// Mitsubishi GX Developer project: パレット移載装置   PLC: Q02

PROGRAM ALARM
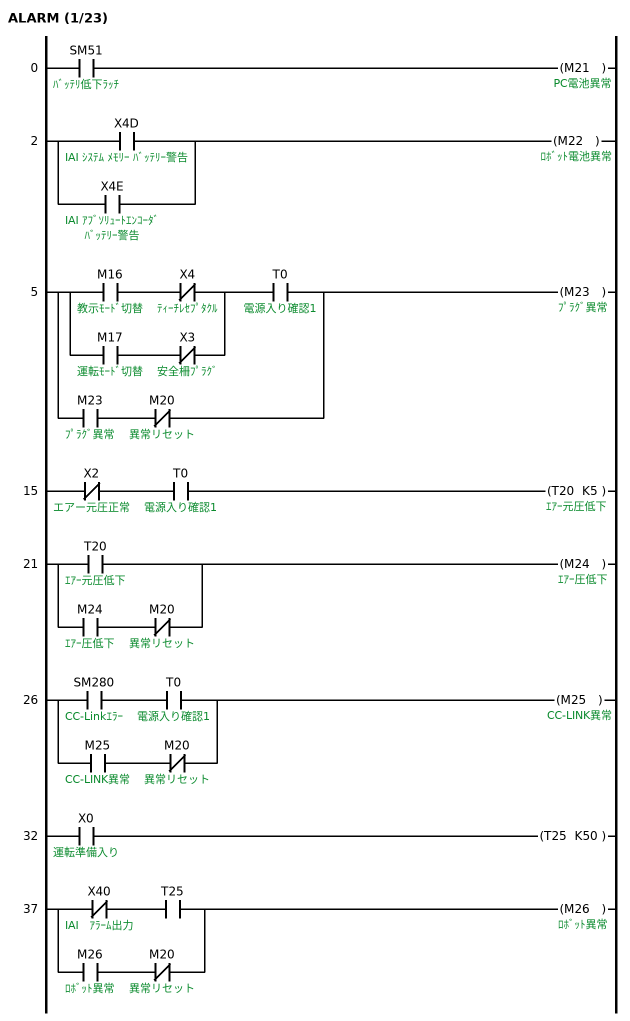
0     LD      SM51  ; ﾊﾞｯﾃﾘ低下ﾗｯﾁ
      OUT     M21  ; PC電池異常
2     LD      X4D  ; IAI ｼｽﾃﾑ ﾒﾓﾘｰ ﾊﾞｯﾃﾘｰ警告
      OR      X4E  ; IAI ｱﾌﾞｿﾘｭｰﾄｴﾝｺｰﾀﾞ ﾊﾞｯﾃﾘｰ警告
      OUT     M22  ; ﾛﾎﾞｯﾄ電池異常
5     LD      M16  ; 教示ﾓｰﾄﾞ切替
      ANI     X4  ; ﾃｨｰﾁﾚｾﾌﾟﾀｸﾙ
      LD      M17  ; 運転ﾓｰﾄﾞ切替
      ANI     X3  ; 安全柵ﾌﾟﾗｸﾞ
      ORB
      AND     T0  ; 電源入り確認1
      LD      M23  ; ﾌﾟﾗｸﾞ異常
      ANI     M20  ; 異常リセット
      ORB
      OUT     M23  ; ﾌﾟﾗｸﾞ異常
15    LDI     X2  ; エアー元圧正常
      AND     T0  ; 電源入り確認1
      OUT     T20 K5  ; ｴｱｰ元圧低下
21    LD      T20  ; ｴｱｰ元圧低下
      LD      M24  ; ｴｱｰ圧低下
      ANI     M20  ; 異常リセット
      ORB
      OUT     M24  ; ｴｱｰ圧低下
26    LD      SM280  ; CC-Linkｴﾗｰ
      AND     T0  ; 電源入り確認1
      LD      M25  ; CC-LINK異常
      ANI     M20  ; 異常リセット
      ORB
      OUT     M25  ; CC-LINK異常
32    LD      X0  ; 運転準備入り
      OUT     T25 K50
37    LDI     X40  ; IAI　ｱﾗｰﾑ出力
      AND     T25
      LD      M26  ; ﾛﾎﾞｯﾄ異常
      ANI     M20  ; 異常リセット
      ORB
      OUT     M26  ; ﾛﾎﾞｯﾄ異常
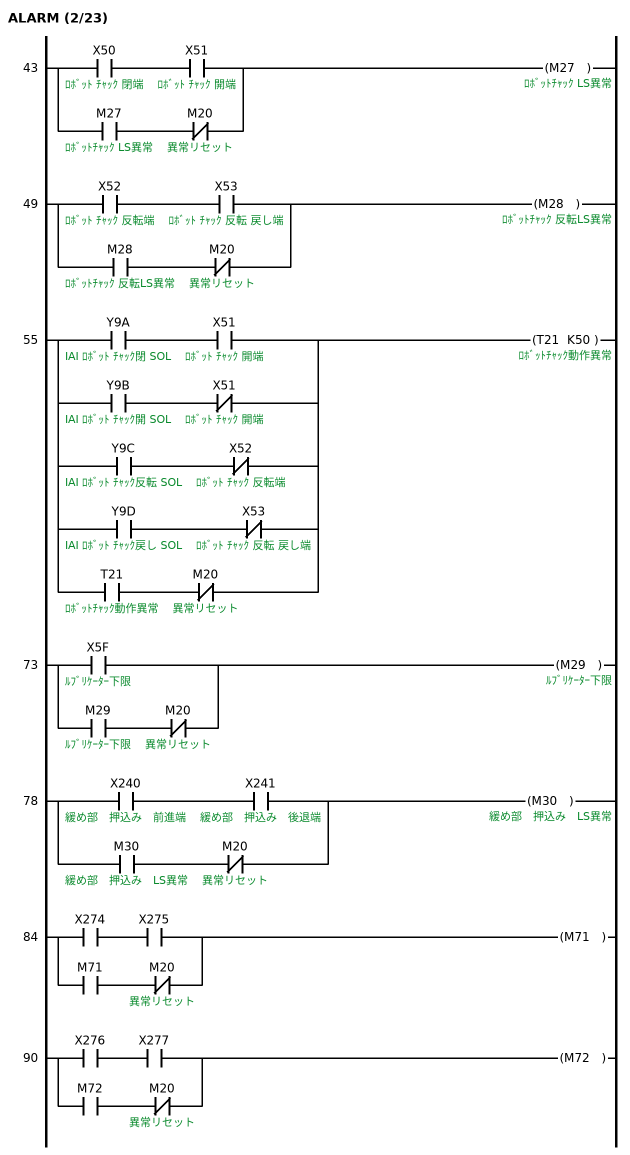
43    LD      X50  ; ﾛﾎﾞｯﾄ ﾁｬｯｸ 閉端
      AND     X51  ; ﾛﾎﾞｯﾄ ﾁｬｯｸ 開端
      LD      M27  ; ﾛﾎﾞｯﾄﾁｬｯｸ LS異常
      ANI     M20  ; 異常リセット
      ORB
      OUT     M27  ; ﾛﾎﾞｯﾄﾁｬｯｸ LS異常
49    LD      X52  ; ﾛﾎﾞｯﾄ ﾁｬｯｸ 反転端
      AND     X53  ; ﾛﾎﾞｯﾄ ﾁｬｯｸ 反転 戻し端
      LD      M28  ; ﾛﾎﾞｯﾄﾁｬｯｸ 反転LS異常
      ANI     M20  ; 異常リセット
      ORB
      OUT     M28  ; ﾛﾎﾞｯﾄﾁｬｯｸ 反転LS異常
55    LD      Y9A  ; IAI ﾛﾎﾞｯﾄ ﾁｬｯｸ閉 SOL
      AND     X51  ; ﾛﾎﾞｯﾄ ﾁｬｯｸ 開端
      LD      Y9B  ; IAI ﾛﾎﾞｯﾄ ﾁｬｯｸ開 SOL
      ANI     X51  ; ﾛﾎﾞｯﾄ ﾁｬｯｸ 開端
      ORB
      LD      Y9C  ; IAI ﾛﾎﾞｯﾄ ﾁｬｯｸ反転 SOL
      ANI     X52  ; ﾛﾎﾞｯﾄ ﾁｬｯｸ 反転端
      ORB
      LD      Y9D  ; IAI ﾛﾎﾞｯﾄ ﾁｬｯｸ戻し SOL
      ANI     X53  ; ﾛﾎﾞｯﾄ ﾁｬｯｸ 反転 戻し端
      ORB
      LD      T21  ; ﾛﾎﾞｯﾄﾁｬｯｸ動作異常
      ANI     M20  ; 異常リセット
      ORB
      OUT     T21 K50  ; ﾛﾎﾞｯﾄﾁｬｯｸ動作異常
73    LD      X5F  ; ﾙﾌﾞﾘｹｰﾀｰ下限
      LD      M29  ; ﾙﾌﾞﾘｹｰﾀｰ下限
      ANI     M20  ; 異常リセット
      ORB
      OUT     M29  ; ﾙﾌﾞﾘｹｰﾀｰ下限
78    LD      X240  ; 緩め部　押込み　前進端
      AND     X241  ; 緩め部　押込み　後退端
      LD      M30  ; 緩め部　押込み　LS異常
      ANI     M20  ; 異常リセット
      ORB
      OUT     M30  ; 緩め部　押込み　LS異常
84    LD      X274
      AND     X275
      LD      M71
      ANI     M20  ; 異常リセット
      ORB
      OUT     M71
90    LD      X276
      AND     X277
      LD      M72
      ANI     M20  ; 異常リセット
      ORB
      OUT     M72
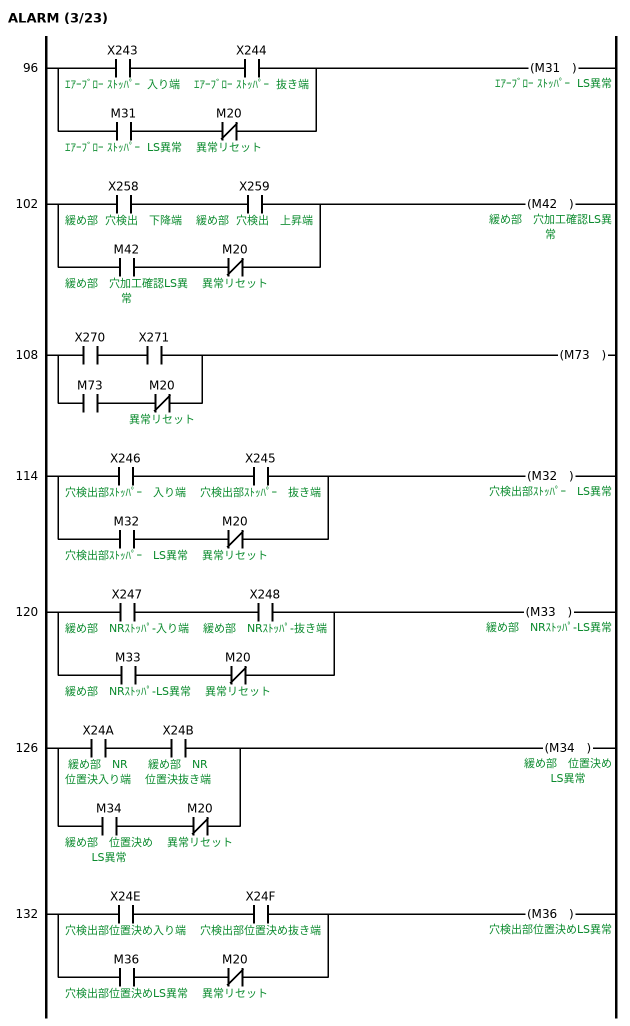
96    LD      X243  ; ｴｱｰﾌﾞﾛｰ ｽﾄｯﾊﾟｰ  入り端
      AND     X244  ; ｴｱｰﾌﾞﾛｰ ｽﾄｯﾊﾟｰ  抜き端
      LD      M31  ; ｴｱｰﾌﾞﾛｰ ｽﾄｯﾊﾟｰ  LS異常
      ANI     M20  ; 異常リセット
      ORB
      OUT     M31  ; ｴｱｰﾌﾞﾛｰ ｽﾄｯﾊﾟｰ  LS異常
102   LD      X258  ; 緩め部  穴検出　下降端
      AND     X259  ; 緩め部  穴検出　上昇端
      LD      M42  ; 緩め部　穴加工確認LS異常
      ANI     M20  ; 異常リセット
      ORB
      OUT     M42  ; 緩め部　穴加工確認LS異常
108   LD      X270
      AND     X271
      LD      M73
      ANI     M20  ; 異常リセット
      ORB
      OUT     M73
114   LD      X246  ; 穴検出部ｽﾄｯﾊﾟｰ　入り端
      AND     X245  ; 穴検出部ｽﾄｯﾊﾟｰ　抜き端
      LD      M32  ; 穴検出部ｽﾄｯﾊﾟｰ　LS異常
      ANI     M20  ; 異常リセット
      ORB
      OUT     M32  ; 穴検出部ｽﾄｯﾊﾟｰ　LS異常
120   LD      X247  ; 緩め部　NRｽﾄｯﾊﾟ-入り端
      AND     X248  ; 緩め部　NRｽﾄｯﾊﾟ-抜き端
      LD      M33  ; 緩め部　NRｽﾄｯﾊﾟ-LS異常
      ANI     M20  ; 異常リセット
      ORB
      OUT     M33  ; 緩め部　NRｽﾄｯﾊﾟ-LS異常
126   LD      X24A  ; 緩め部　NR 位置決入り端
      AND     X24B  ; 緩め部　NR 位置決抜き端
      LD      M34  ; 緩め部　位置決め LS異常
      ANI     M20  ; 異常リセット
      ORB
      OUT     M34  ; 緩め部　位置決め LS異常
132   LD      X24E  ; 穴検出部位置決め入り端
      AND     X24F  ; 穴検出部位置決め抜き端
      LD      M36  ; 穴検出部位置決めLS異常
      ANI     M20  ; 異常リセット
      ORB
      OUT     M36  ; 穴検出部位置決めLS異常
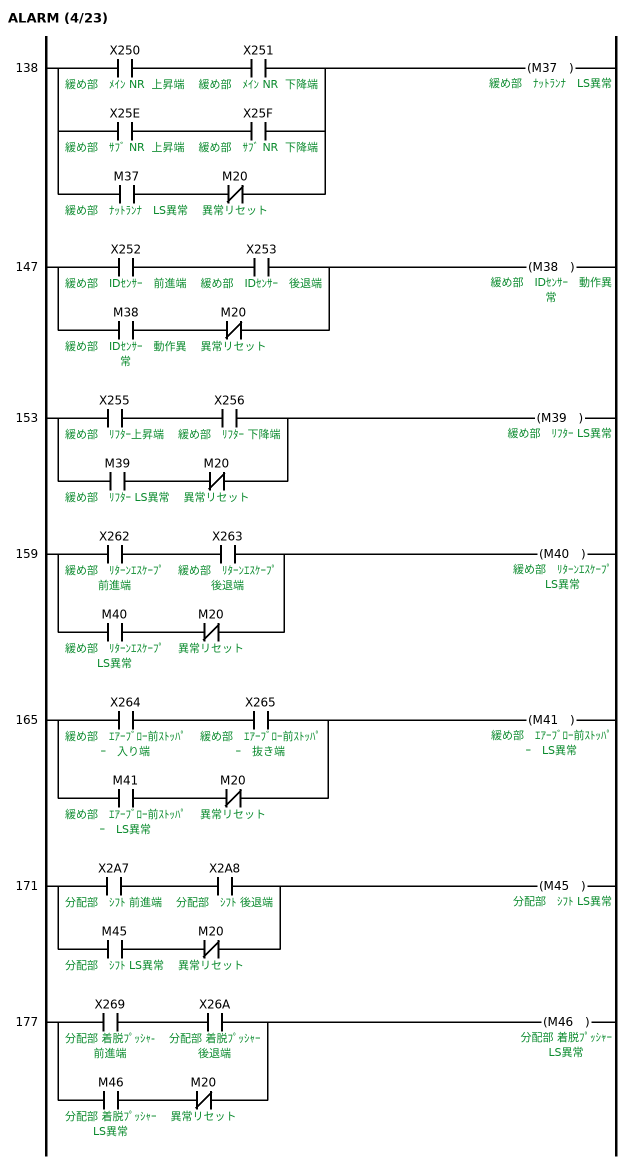
138   LD      X250  ; 緩め部　ﾒｲﾝ NR  上昇端
      AND     X251  ; 緩め部　ﾒｲﾝ NR  下降端
      LD      X25E  ; 緩め部　ｻﾌﾞ NR  上昇端
      AND     X25F  ; 緩め部　ｻﾌﾞ NR  下降端
      ORB
      LD      M37  ; 緩め部　ﾅｯﾄﾗﾝﾅ　LS異常
      ANI     M20  ; 異常リセット
      ORB
      OUT     M37  ; 緩め部　ﾅｯﾄﾗﾝﾅ　LS異常
147   LD      X252  ; 緩め部　IDｾﾝｻｰ　前進端
      AND     X253  ; 緩め部　IDｾﾝｻｰ　後退端
      LD      M38  ; 緩め部　IDｾﾝｻｰ　動作異常
      ANI     M20  ; 異常リセット
      ORB
      OUT     M38  ; 緩め部　IDｾﾝｻｰ　動作異常
153   LD      X255  ; 緩め部　ﾘﾌﾀｰ上昇端
      AND     X256  ; 緩め部　ﾘﾌﾀｰ 下降端
      LD      M39  ; 緩め部　ﾘﾌﾀｰ LS異常
      ANI     M20  ; 異常リセット
      ORB
      OUT     M39  ; 緩め部　ﾘﾌﾀｰ LS異常
159   LD      X262  ; 緩め部　ﾘﾀｰﾝｴｽｹｰﾌﾟ 前進端
      AND     X263  ; 緩め部　ﾘﾀｰﾝｴｽｹｰﾌﾟ 後退端
      LD      M40  ; 緩め部　ﾘﾀｰﾝｴｽｹｰﾌﾟ LS異常
      ANI     M20  ; 異常リセット
      ORB
      OUT     M40  ; 緩め部　ﾘﾀｰﾝｴｽｹｰﾌﾟ LS異常
165   LD      X264  ; 緩め部　ｴｱｰﾌﾞﾛｰ前ｽﾄｯﾊﾟｰ　入り端
      AND     X265  ; 緩め部　ｴｱｰﾌﾞﾛｰ前ｽﾄｯﾊﾟｰ　抜き端
      LD      M41  ; 緩め部　ｴｱｰﾌﾞﾛｰ前ｽﾄｯﾊﾟｰ　LS異常
      ANI     M20  ; 異常リセット
      ORB
      OUT     M41  ; 緩め部　ｴｱｰﾌﾞﾛｰ前ｽﾄｯﾊﾟｰ　LS異常
171   LD      X2A7  ; 分配部　ｼﾌﾄ 前進端
      AND     X2A8  ; 分配部　ｼﾌﾄ 後退端
      LD      M45  ; 分配部　ｼﾌﾄ LS異常
      ANI     M20  ; 異常リセット
      ORB
      OUT     M45  ; 分配部　ｼﾌﾄ LS異常
177   LD      X269  ; 分配部 着脱ﾌﾟｯｼｬ- 前進端
      AND     X26A  ; 分配部 着脱ﾌﾟｯｼｬｰ 後退端
      LD      M46  ; 分配部 着脱ﾌﾟｯｼｬｰ LS異常
      ANI     M20  ; 異常リセット
      ORB
      OUT     M46  ; 分配部 着脱ﾌﾟｯｼｬｰ LS異常
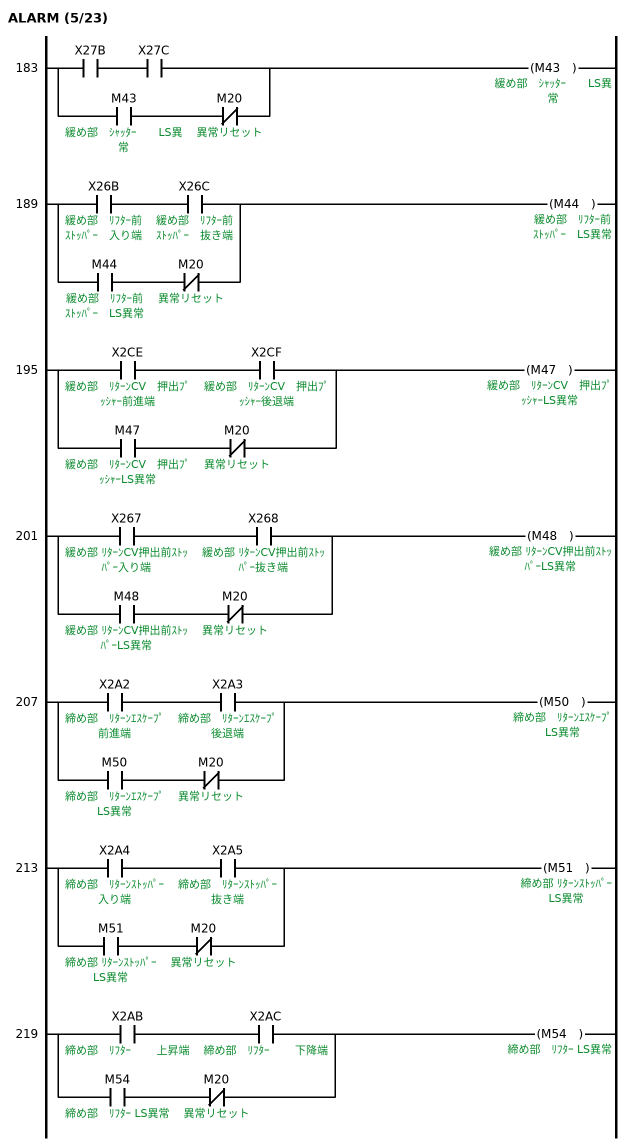
183   LD      X27B
      AND     X27C
      LD      M43  ; 緩め部　ｼｬｯﾀｰ　　LS異常
      ANI     M20  ; 異常リセット
      ORB
      OUT     M43  ; 緩め部　ｼｬｯﾀｰ　　LS異常
189   LD      X26B  ; 緩め部　ﾘﾌﾀｰ前  ｽﾄｯﾊﾟｰ　入り端
      AND     X26C  ; 緩め部　ﾘﾌﾀｰ前  ｽﾄｯﾊﾟｰ　抜き端
      LD      M44  ; 緩め部　ﾘﾌﾀｰ前  ｽﾄｯﾊﾟｰ　LS異常
      ANI     M20  ; 異常リセット
      ORB
      OUT     M44  ; 緩め部　ﾘﾌﾀｰ前  ｽﾄｯﾊﾟｰ　LS異常
195   LD      X2CE  ; 緩め部　ﾘﾀｰﾝCV　押出ﾌﾟｯｼｬｰ前進端
      AND     X2CF  ; 緩め部　ﾘﾀｰﾝCV　押出ﾌﾟｯｼｬｰ後退端
      LD      M47  ; 緩め部　ﾘﾀｰﾝCV　押出ﾌﾟｯｼｬｰLS異常
      ANI     M20  ; 異常リセット
      ORB
      OUT     M47  ; 緩め部　ﾘﾀｰﾝCV　押出ﾌﾟｯｼｬｰLS異常
201   LD      X267  ; 緩め部 ﾘﾀｰﾝCV押出前ｽﾄｯﾊﾟｰ入り端
      AND     X268  ; 緩め部 ﾘﾀｰﾝCV押出前ｽﾄｯﾊﾟｰ抜き端
      LD      M48  ; 緩め部 ﾘﾀｰﾝCV押出前ｽﾄｯﾊﾟｰLS異常
      ANI     M20  ; 異常リセット
      ORB
      OUT     M48  ; 緩め部 ﾘﾀｰﾝCV押出前ｽﾄｯﾊﾟｰLS異常
207   LD      X2A2  ; 締め部　ﾘﾀｰﾝｴｽｹｰﾌﾟ 前進端
      AND     X2A3  ; 締め部　ﾘﾀｰﾝｴｽｹｰﾌﾟ 後退端
      LD      M50  ; 締め部　ﾘﾀｰﾝｴｽｹｰﾌﾟ LS異常
      ANI     M20  ; 異常リセット
      ORB
      OUT     M50  ; 締め部　ﾘﾀｰﾝｴｽｹｰﾌﾟ LS異常
213   LD      X2A4  ; 締め部　ﾘﾀｰﾝｽﾄｯﾊﾟｰ 入り端
      AND     X2A5  ; 締め部　ﾘﾀｰﾝｽﾄｯﾊﾟｰ 抜き端
      LD      M51  ; 締め部 ﾘﾀｰﾝｽﾄｯﾊﾟｰ LS異常
      ANI     M20  ; 異常リセット
      ORB
      OUT     M51  ; 締め部 ﾘﾀｰﾝｽﾄｯﾊﾟｰ LS異常
219   LD      X2AB  ; 締め部　ﾘﾌﾀｰ 　　上昇端
      AND     X2AC  ; 締め部　ﾘﾌﾀｰ 　　下降端
      LD      M54  ; 締め部　ﾘﾌﾀｰ LS異常
      ANI     M20  ; 異常リセット
      ORB
      OUT     M54  ; 締め部　ﾘﾌﾀｰ LS異常
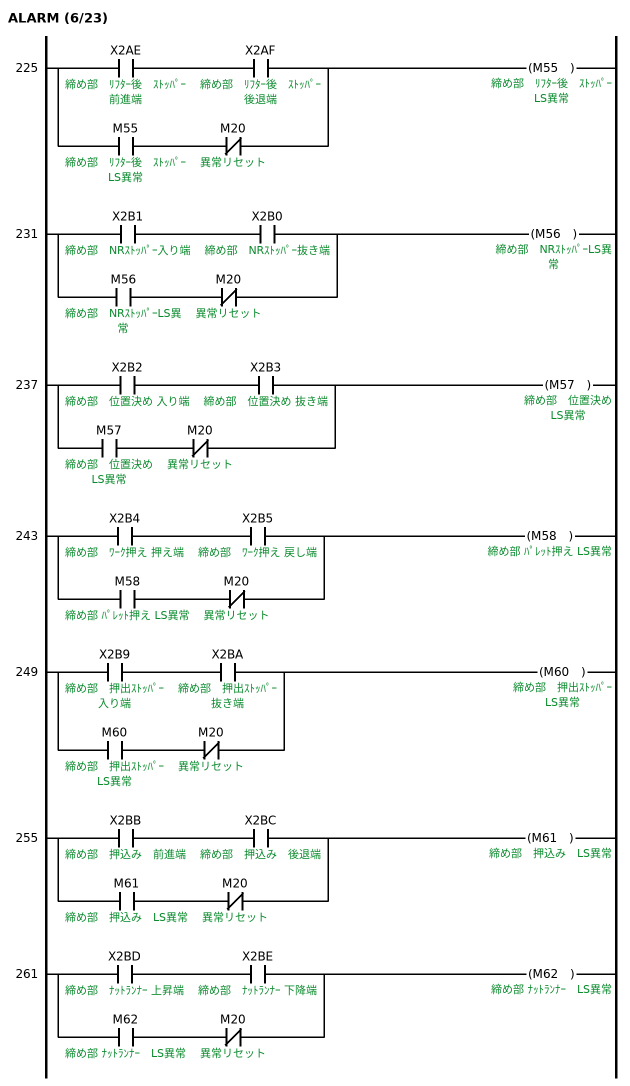
225   LD      X2AE  ; 締め部　ﾘﾌﾀｰ後　ｽﾄｯﾊﾟｰ　前進端
      AND     X2AF  ; 締め部　ﾘﾌﾀｰ後　ｽﾄｯﾊﾟｰ　後退端
      LD      M55  ; 締め部　ﾘﾌﾀｰ後　ｽﾄｯﾊﾟｰ　LS異常
      ANI     M20  ; 異常リセット
      ORB
      OUT     M55  ; 締め部　ﾘﾌﾀｰ後　ｽﾄｯﾊﾟｰ　LS異常
231   LD      X2B1  ; 締め部　NRｽﾄｯﾊﾟｰ入り端
      AND     X2B0  ; 締め部　NRｽﾄｯﾊﾟｰ抜き端
      LD      M56  ; 締め部　NRｽﾄｯﾊﾟｰLS異常
      ANI     M20  ; 異常リセット
      ORB
      OUT     M56  ; 締め部　NRｽﾄｯﾊﾟｰLS異常
237   LD      X2B2  ; 締め部　位置決め 入り端
      AND     X2B3  ; 締め部　位置決め 抜き端
      LD      M57  ; 締め部　位置決め LS異常
      ANI     M20  ; 異常リセット
      ORB
      OUT     M57  ; 締め部　位置決め LS異常
243   LD      X2B4  ; 締め部　ﾜｰｸ押え 押え端
      AND     X2B5  ; 締め部　ﾜｰｸ押え 戻し端
      LD      M58  ; 締め部 ﾊﾟﾚｯﾄ押え LS異常
      ANI     M20  ; 異常リセット
      ORB
      OUT     M58  ; 締め部 ﾊﾟﾚｯﾄ押え LS異常
249   LD      X2B9  ; 締め部　押出ｽﾄｯﾊﾟｰ 入り端
      AND     X2BA  ; 締め部　押出ｽﾄｯﾊﾟｰ 抜き端
      LD      M60  ; 締め部　押出ｽﾄｯﾊﾟｰ LS異常
      ANI     M20  ; 異常リセット
      ORB
      OUT     M60  ; 締め部　押出ｽﾄｯﾊﾟｰ LS異常
255   LD      X2BB  ; 締め部　押込み　前進端
      AND     X2BC  ; 締め部　押込み　後退端
      LD      M61  ; 締め部　押込み　LS異常
      ANI     M20  ; 異常リセット
      ORB
      OUT     M61  ; 締め部　押込み　LS異常
261   LD      X2BD  ; 締め部　ﾅｯﾄﾗﾝﾅｰ 上昇端
      AND     X2BE  ; 締め部　ﾅｯﾄﾗﾝﾅｰ 下降端
      LD      M62  ; 締め部 ﾅｯﾄﾗﾝﾅｰ　LS異常
      ANI     M20  ; 異常リセット
      ORB
      OUT     M62  ; 締め部 ﾅｯﾄﾗﾝﾅｰ　LS異常
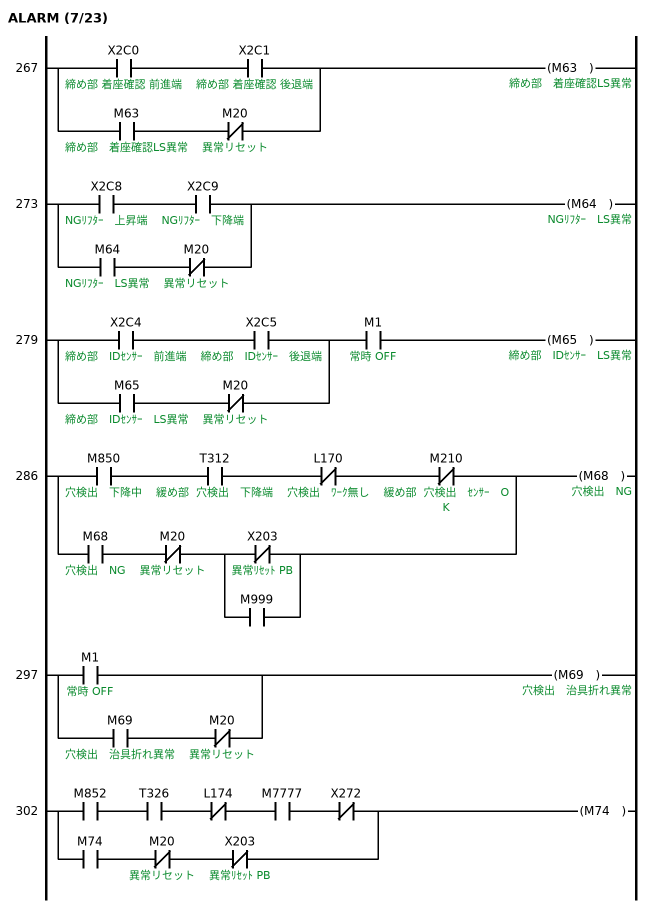
267   LD      X2C0  ; 締め部 着座確認 前進端
      AND     X2C1  ; 締め部 着座確認 後退端
      LD      M63  ; 締め部　着座確認LS異常
      ANI     M20  ; 異常リセット
      ORB
      OUT     M63  ; 締め部　着座確認LS異常
273   LD      X2C8  ; NGﾘﾌﾀｰ　上昇端
      AND     X2C9  ; NGﾘﾌﾀｰ　下降端
      LD      M64  ; NGﾘﾌﾀｰ　LS異常
      ANI     M20  ; 異常リセット
      ORB
      OUT     M64  ; NGﾘﾌﾀｰ　LS異常
279   LD      X2C4  ; 締め部　IDｾﾝｻｰ　前進端
      AND     X2C5  ; 締め部　IDｾﾝｻｰ　後退端
      LD      M65  ; 締め部　IDｾﾝｻｰ　LS異常
      ANI     M20  ; 異常リセット
      ORB
      AND     M1  ; 常時 OFF
      OUT     M65  ; 締め部　IDｾﾝｻｰ　LS異常
286   LD      M850  ; 穴検出　下降中
      AND     T312  ; 緩め部  穴検出　下降端
      ANI     L170  ; 穴検出　ﾜｰｸ無し
      ANI     M210  ; 緩め部  穴検出　ｾﾝｻｰ　OK
      LD      M68  ; 穴検出　NG
      ANI     M20  ; 異常リセット
      LDI     X203  ; 異常ﾘｾｯﾄ PB
      OR      M999
      ANB
      ORB
      OUT     M68  ; 穴検出　NG
297   LD      M1  ; 常時 OFF
      LD      M69  ; 穴検出　治具折れ異常
      ANI     M20  ; 異常リセット
      ORB
      OUT     M69  ; 穴検出　治具折れ異常
302   LD      M852
      AND     T326
      ANI     L174
      AND     M7777
      ANI     X272
      LD      M74
      ANI     M20  ; 異常リセット
      ANI     X203  ; 異常ﾘｾｯﾄ PB
      ORB
      OUT     M74
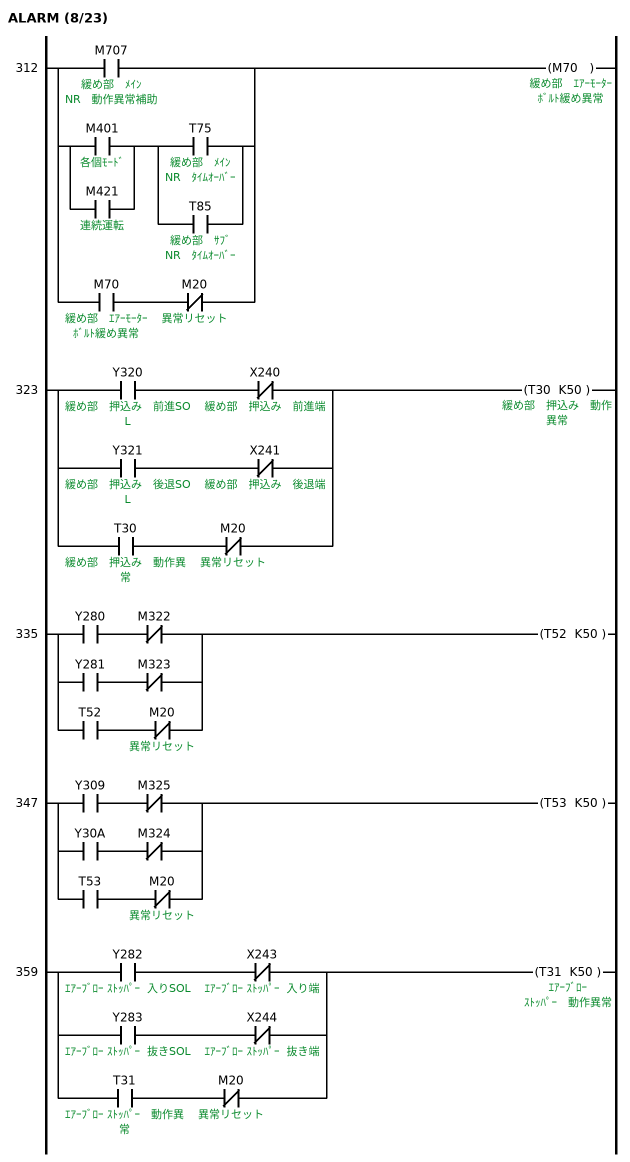
312   LD      M707  ; 緩め部　ﾒｲﾝ NR　動作異常補助
      LD      M401  ; 各個ﾓｰﾄﾞ
      OR      M421  ; 連続運転
      LD      T75  ; 緩め部　ﾒｲﾝ NR　ﾀｲﾑｵｰﾊﾞｰ
      OR      T85  ; 緩め部　ｻﾌﾞ NR　ﾀｲﾑｵｰﾊﾞｰ
      ANB
      ORB
      LD      M70  ; 緩め部　ｴｱｰﾓｰﾀｰ ﾎﾞﾙﾄ緩め異常
      ANI     M20  ; 異常リセット
      ORB
      OUT     M70  ; 緩め部　ｴｱｰﾓｰﾀｰ ﾎﾞﾙﾄ緩め異常
323   LD      Y320  ; 緩め部　押込み　前進SOL
      ANI     X240  ; 緩め部　押込み　前進端
      LD      Y321  ; 緩め部　押込み　後退SOL
      ANI     X241  ; 緩め部　押込み　後退端
      ORB
      LD      T30  ; 緩め部　押込み　動作異常
      ANI     M20  ; 異常リセット
      ORB
      OUT     T30 K50  ; 緩め部　押込み　動作異常
335   LD      Y280
      ANI     M322
      LD      Y281
      ANI     M323
      ORB
      LD      T52
      ANI     M20  ; 異常リセット
      ORB
      OUT     T52 K50
347   LD      Y309
      ANI     M325
      LD      Y30A
      ANI     M324
      ORB
      LD      T53
      ANI     M20  ; 異常リセット
      ORB
      OUT     T53 K50
359   LD      Y282  ; ｴｱｰﾌﾞﾛｰ ｽﾄｯﾊﾟｰ  入りSOL
      ANI     X243  ; ｴｱｰﾌﾞﾛｰ ｽﾄｯﾊﾟｰ  入り端
      LD      Y283  ; ｴｱｰﾌﾞﾛｰ ｽﾄｯﾊﾟｰ  抜きSOL
      ANI     X244  ; ｴｱｰﾌﾞﾛｰ ｽﾄｯﾊﾟｰ  抜き端
      ORB
      LD      T31  ; ｴｱｰﾌﾞﾛｰ ｽﾄｯﾊﾟｰ　動作異常
      ANI     M20  ; 異常リセット
      ORB
      OUT     T31 K50  ; ｴｱｰﾌﾞﾛｰ ｽﾄｯﾊﾟｰ　動作異常
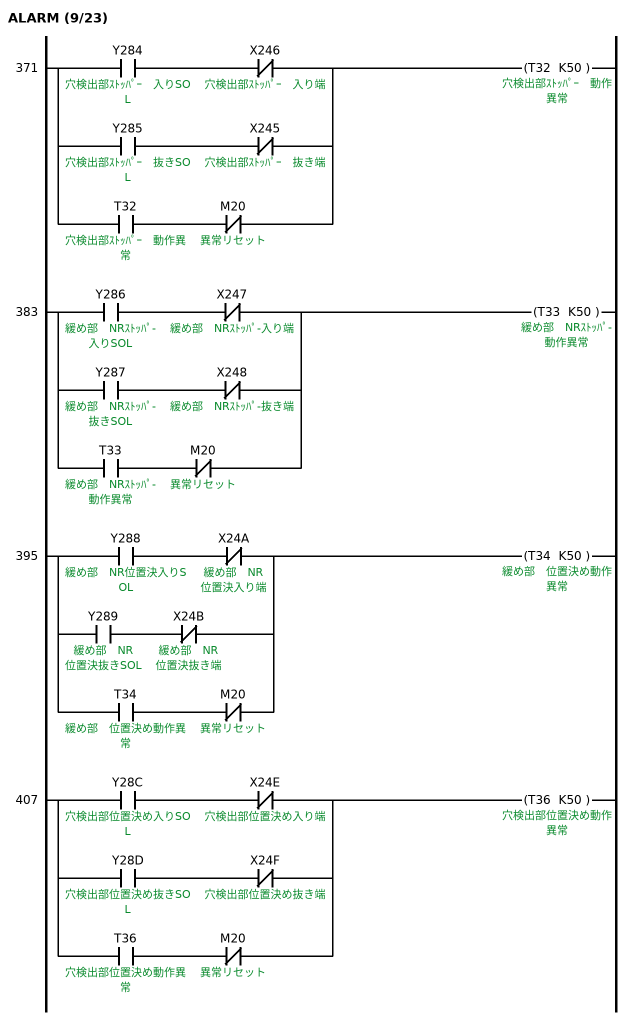
371   LD      Y284  ; 穴検出部ｽﾄｯﾊﾟｰ　入りSOL
      ANI     X246  ; 穴検出部ｽﾄｯﾊﾟｰ　入り端
      LD      Y285  ; 穴検出部ｽﾄｯﾊﾟｰ　抜きSOL
      ANI     X245  ; 穴検出部ｽﾄｯﾊﾟｰ　抜き端
      ORB
      LD      T32  ; 穴検出部ｽﾄｯﾊﾟｰ　動作異常
      ANI     M20  ; 異常リセット
      ORB
      OUT     T32 K50  ; 穴検出部ｽﾄｯﾊﾟｰ　動作異常
383   LD      Y286  ; 緩め部　NRｽﾄｯﾊﾟ-入りSOL
      ANI     X247  ; 緩め部　NRｽﾄｯﾊﾟ-入り端
      LD      Y287  ; 緩め部　NRｽﾄｯﾊﾟ-抜きSOL
      ANI     X248  ; 緩め部　NRｽﾄｯﾊﾟ-抜き端
      ORB
      LD      T33  ; 緩め部　NRｽﾄｯﾊﾟ-動作異常
      ANI     M20  ; 異常リセット
      ORB
      OUT     T33 K50  ; 緩め部　NRｽﾄｯﾊﾟ-動作異常
395   LD      Y288  ; 緩め部　NR位置決入りSOL
      ANI     X24A  ; 緩め部　NR 位置決入り端
      LD      Y289  ; 緩め部　NR 位置決抜きSOL
      ANI     X24B  ; 緩め部　NR 位置決抜き端
      ORB
      LD      T34  ; 緩め部　位置決め動作異常
      ANI     M20  ; 異常リセット
      ORB
      OUT     T34 K50  ; 緩め部　位置決め動作異常
407   LD      Y28C  ; 穴検出部位置決め入りSOL
      ANI     X24E  ; 穴検出部位置決め入り端
      LD      Y28D  ; 穴検出部位置決め抜きSOL
      ANI     X24F  ; 穴検出部位置決め抜き端
      ORB
      LD      T36  ; 穴検出部位置決め動作異常
      ANI     M20  ; 異常リセット
      ORB
      OUT     T36 K50  ; 穴検出部位置決め動作異常
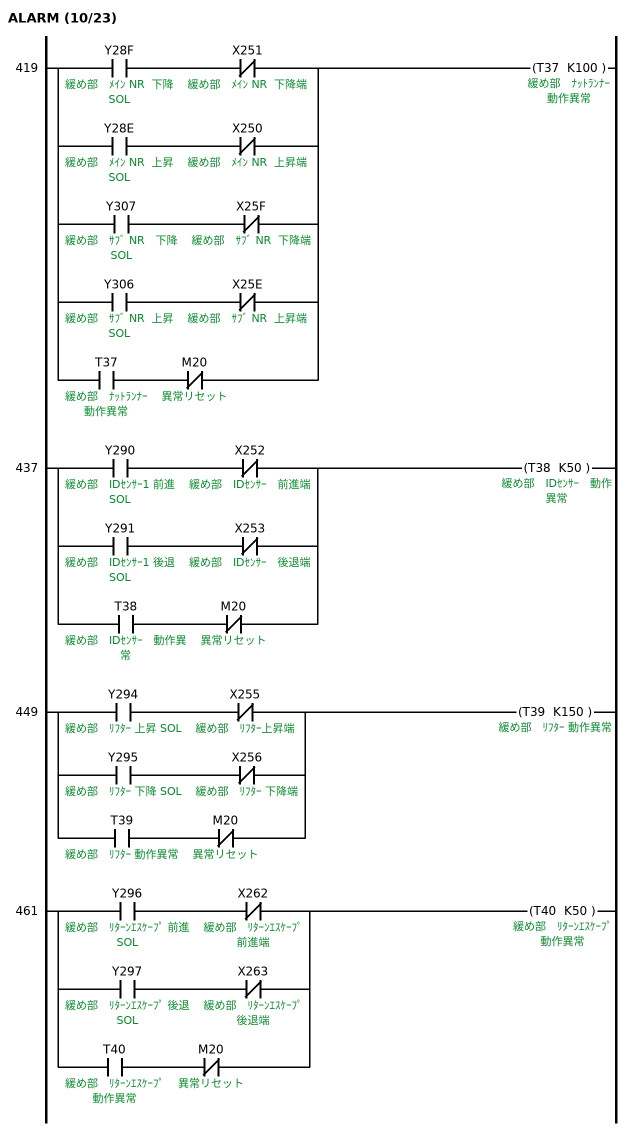
419   LD      Y28F  ; 緩め部　ﾒｲﾝ NR  下降 SOL
      ANI     X251  ; 緩め部　ﾒｲﾝ NR  下降端
      LD      Y28E  ; 緩め部　ﾒｲﾝ NR  上昇 SOL
      ANI     X250  ; 緩め部　ﾒｲﾝ NR  上昇端
      ORB
      LD      Y307  ; 緩め部　ｻﾌﾞ NR　下降 SOL
      ANI     X25F  ; 緩め部　ｻﾌﾞ NR  下降端
      ORB
      LD      Y306  ; 緩め部　ｻﾌﾞ NR  上昇 SOL
      ANI     X25E  ; 緩め部　ｻﾌﾞ NR  上昇端
      ORB
      LD      T37  ; 緩め部　ﾅｯﾄﾗﾝﾅｰ 動作異常
      ANI     M20  ; 異常リセット
      ORB
      OUT     T37 K100  ; 緩め部　ﾅｯﾄﾗﾝﾅｰ 動作異常
437   LD      Y290  ; 緩め部　IDｾﾝｻｰ1 前進 SOL
      ANI     X252  ; 緩め部　IDｾﾝｻｰ　前進端
      LD      Y291  ; 緩め部　IDｾﾝｻｰ1 後退 SOL
      ANI     X253  ; 緩め部　IDｾﾝｻｰ　後退端
      ORB
      LD      T38  ; 緩め部　IDｾﾝｻｰ　動作異常
      ANI     M20  ; 異常リセット
      ORB
      OUT     T38 K50  ; 緩め部　IDｾﾝｻｰ　動作異常
449   LD      Y294  ; 緩め部　ﾘﾌﾀｰ 上昇 SOL
      ANI     X255  ; 緩め部　ﾘﾌﾀｰ上昇端
      LD      Y295  ; 緩め部　ﾘﾌﾀｰ 下降 SOL
      ANI     X256  ; 緩め部　ﾘﾌﾀｰ 下降端
      ORB
      LD      T39  ; 緩め部　ﾘﾌﾀｰ 動作異常
      ANI     M20  ; 異常リセット
      ORB
      OUT     T39 K150  ; 緩め部　ﾘﾌﾀｰ 動作異常
461   LD      Y296  ; 緩め部　ﾘﾀｰﾝｴｽｹｰﾌﾟ 前進 SOL
      ANI     X262  ; 緩め部　ﾘﾀｰﾝｴｽｹｰﾌﾟ 前進端
      LD      Y297  ; 緩め部　ﾘﾀｰﾝｴｽｹｰﾌﾟ 後退 SOL
      ANI     X263  ; 緩め部　ﾘﾀｰﾝｴｽｹｰﾌﾟ 後退端
      ORB
      LD      T40  ; 緩め部　ﾘﾀｰﾝｴｽｹｰﾌﾟ 動作異常
      ANI     M20  ; 異常リセット
      ORB
      OUT     T40 K50  ; 緩め部　ﾘﾀｰﾝｴｽｹｰﾌﾟ 動作異常
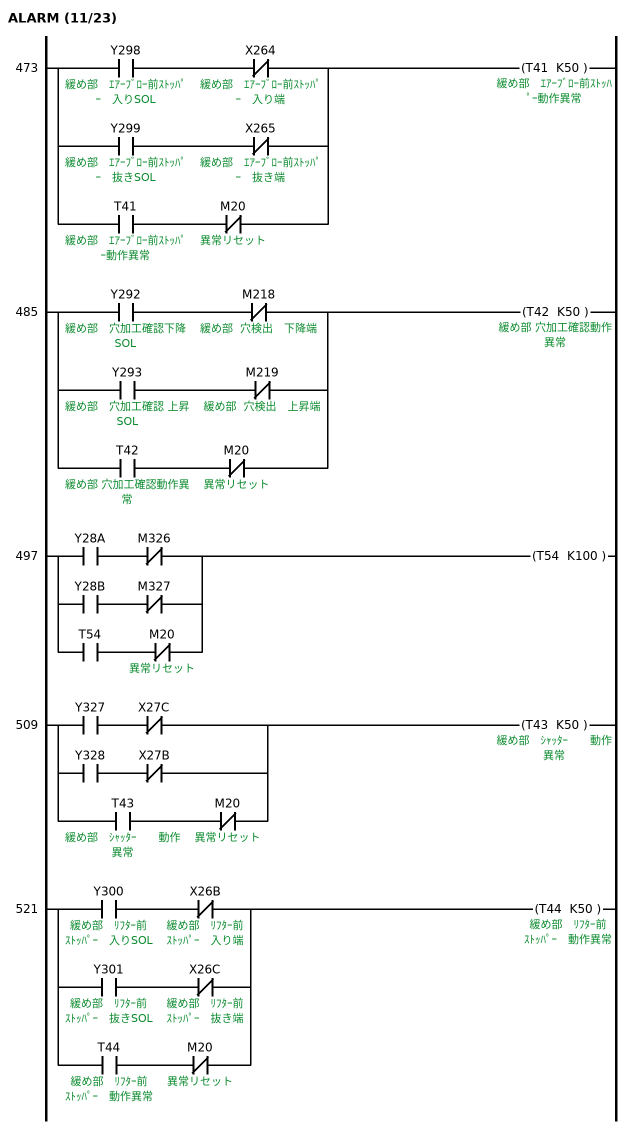
473   LD      Y298  ; 緩め部　ｴｱｰﾌﾞﾛｰ前ｽﾄｯﾊﾟｰ　入りSOL
      ANI     X264  ; 緩め部　ｴｱｰﾌﾞﾛｰ前ｽﾄｯﾊﾟｰ　入り端
      LD      Y299  ; 緩め部　ｴｱｰﾌﾞﾛｰ前ｽﾄｯﾊﾟｰ　抜きSOL
      ANI     X265  ; 緩め部　ｴｱｰﾌﾞﾛｰ前ｽﾄｯﾊﾟｰ　抜き端
      ORB
      LD      T41  ; 緩め部　ｴｱｰﾌﾞﾛｰ前ｽﾄｯﾊﾟｰ動作異常
      ANI     M20  ; 異常リセット
      ORB
      OUT     T41 K50  ; 緩め部　ｴｱｰﾌﾞﾛｰ前ｽﾄｯﾊﾟｰ動作異常
485   LD      Y292  ; 緩め部　穴加工確認下降 SOL
      ANI     M218  ; 緩め部  穴検出　下降端
      LD      Y293  ; 緩め部　穴加工確認 上昇 SOL
      ANI     M219  ; 緩め部  穴検出　上昇端
      ORB
      LD      T42  ; 緩め部 穴加工確認動作異常
      ANI     M20  ; 異常リセット
      ORB
      OUT     T42 K50  ; 緩め部 穴加工確認動作異常
497   LD      Y28A
      ANI     M326
      LD      Y28B
      ANI     M327
      ORB
      LD      T54
      ANI     M20  ; 異常リセット
      ORB
      OUT     T54 K100
509   LD      Y327
      ANI     X27C
      LD      Y328
      ANI     X27B
      ORB
      LD      T43  ; 緩め部　ｼｬｯﾀｰ　　動作異常
      ANI     M20  ; 異常リセット
      ORB
      OUT     T43 K50  ; 緩め部　ｼｬｯﾀｰ　　動作異常
521   LD      Y300  ; 緩め部　ﾘﾌﾀｰ前  ｽﾄｯﾊﾟｰ　入りSOL
      ANI     X26B  ; 緩め部　ﾘﾌﾀｰ前  ｽﾄｯﾊﾟｰ　入り端
      LD      Y301  ; 緩め部　ﾘﾌﾀｰ前  ｽﾄｯﾊﾟｰ　抜きSOL
      ANI     X26C  ; 緩め部　ﾘﾌﾀｰ前  ｽﾄｯﾊﾟｰ　抜き端
      ORB
      LD      T44  ; 緩め部　ﾘﾌﾀｰ前  ｽﾄｯﾊﾟｰ　動作異常
      ANI     M20  ; 異常リセット
      ORB
      OUT     T44 K50  ; 緩め部　ﾘﾌﾀｰ前  ｽﾄｯﾊﾟｰ　動作異常
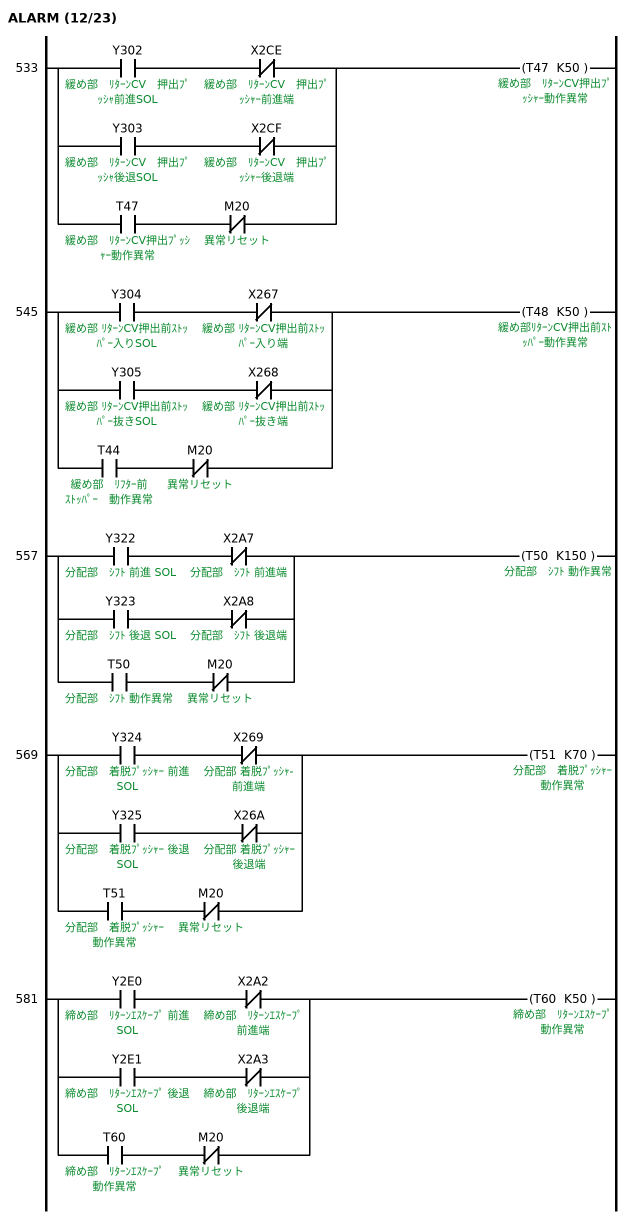
533   LD      Y302  ; 緩め部　ﾘﾀｰﾝCV　押出ﾌﾟｯｼｬ前進SOL
      ANI     X2CE  ; 緩め部　ﾘﾀｰﾝCV　押出ﾌﾟｯｼｬｰ前進端
      LD      Y303  ; 緩め部　ﾘﾀｰﾝCV　押出ﾌﾟｯｼｬ後退SOL
      ANI     X2CF  ; 緩め部　ﾘﾀｰﾝCV　押出ﾌﾟｯｼｬｰ後退端
      ORB
      LD      T47  ; 緩め部　ﾘﾀｰﾝCV押出ﾌﾟｯｼｬｰ動作異常
      ANI     M20  ; 異常リセット
      ORB
      OUT     T47 K50  ; 緩め部　ﾘﾀｰﾝCV押出ﾌﾟｯｼｬｰ動作異常
545   LD      Y304  ; 緩め部 ﾘﾀｰﾝCV押出前ｽﾄｯﾊﾟｰ入りSOL
      ANI     X267  ; 緩め部 ﾘﾀｰﾝCV押出前ｽﾄｯﾊﾟｰ入り端
      LD      Y305  ; 緩め部 ﾘﾀｰﾝCV押出前ｽﾄｯﾊﾟｰ抜きSOL
      ANI     X268  ; 緩め部 ﾘﾀｰﾝCV押出前ｽﾄｯﾊﾟｰ抜き端
      ORB
      LD      T44  ; 緩め部　ﾘﾌﾀｰ前  ｽﾄｯﾊﾟｰ　動作異常
      ANI     M20  ; 異常リセット
      ORB
      OUT     T48 K50  ; 緩め部ﾘﾀｰﾝCV押出前ｽﾄｯﾊﾟｰ動作異常
557   LD      Y322  ; 分配部　ｼﾌﾄ 前進 SOL
      ANI     X2A7  ; 分配部　ｼﾌﾄ 前進端
      LD      Y323  ; 分配部　ｼﾌﾄ 後退 SOL
      ANI     X2A8  ; 分配部　ｼﾌﾄ 後退端
      ORB
      LD      T50  ; 分配部　ｼﾌﾄ 動作異常
      ANI     M20  ; 異常リセット
      ORB
      OUT     T50 K150  ; 分配部　ｼﾌﾄ 動作異常
569   LD      Y324  ; 分配部　着脱ﾌﾟｯｼｬｰ 前進 SOL
      ANI     X269  ; 分配部 着脱ﾌﾟｯｼｬ- 前進端
      LD      Y325  ; 分配部　着脱ﾌﾟｯｼｬｰ 後退 SOL
      ANI     X26A  ; 分配部 着脱ﾌﾟｯｼｬｰ 後退端
      ORB
      LD      T51  ; 分配部　着脱ﾌﾟｯｼｬｰ 動作異常
      ANI     M20  ; 異常リセット
      ORB
      OUT     T51 K70  ; 分配部　着脱ﾌﾟｯｼｬｰ 動作異常
581   LD      Y2E0  ; 締め部　ﾘﾀｰﾝｴｽｹｰﾌﾟ 前進 SOL
      ANI     X2A2  ; 締め部　ﾘﾀｰﾝｴｽｹｰﾌﾟ 前進端
      LD      Y2E1  ; 締め部　ﾘﾀｰﾝｴｽｹｰﾌﾟ 後退 SOL
      ANI     X2A3  ; 締め部　ﾘﾀｰﾝｴｽｹｰﾌﾟ 後退端
      ORB
      LD      T60  ; 締め部　ﾘﾀｰﾝｴｽｹｰﾌﾟ 動作異常
      ANI     M20  ; 異常リセット
      ORB
      OUT     T60 K50  ; 締め部　ﾘﾀｰﾝｴｽｹｰﾌﾟ 動作異常
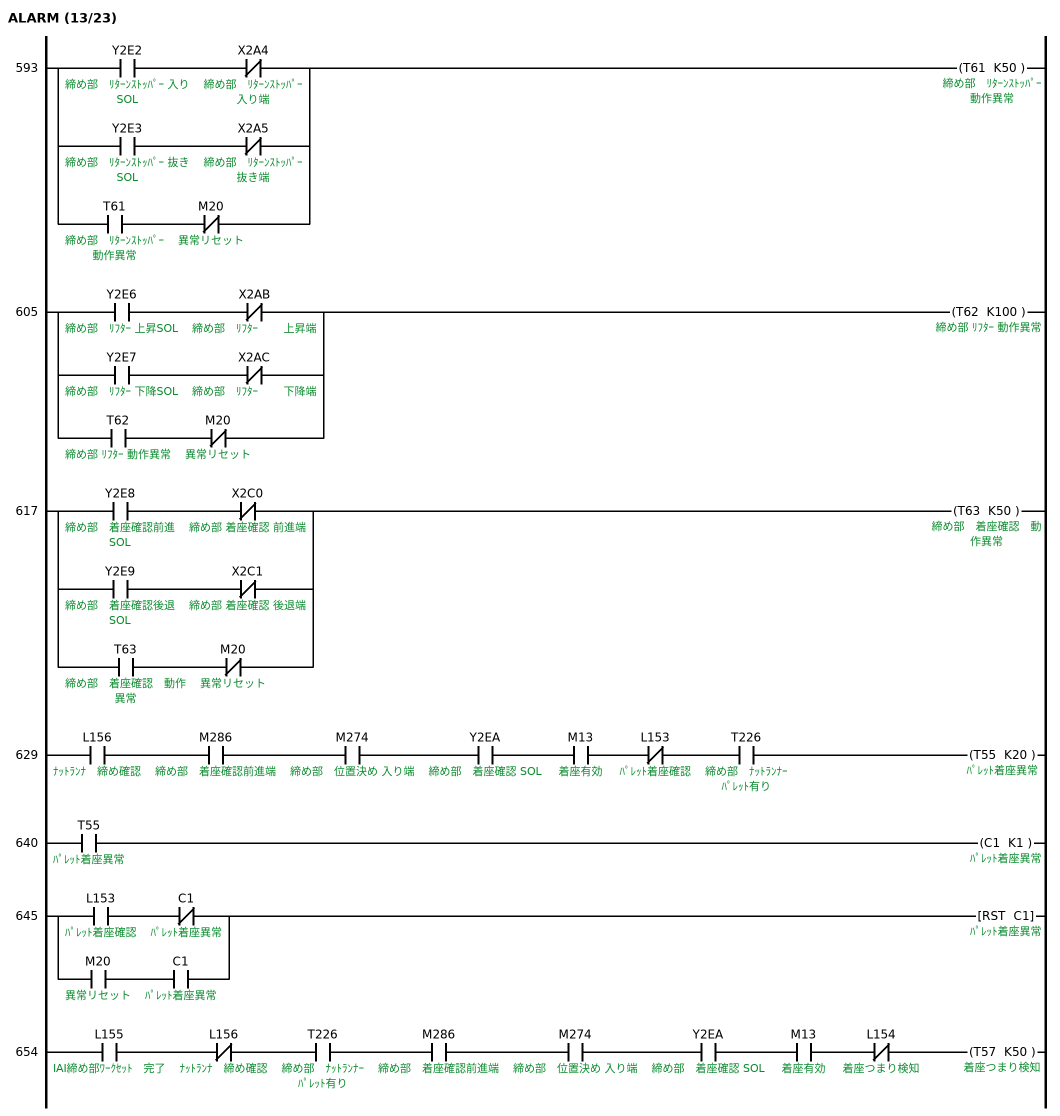
593   LD      Y2E2  ; 締め部　ﾘﾀｰﾝｽﾄｯﾊﾟｰ 入り SOL
      ANI     X2A4  ; 締め部　ﾘﾀｰﾝｽﾄｯﾊﾟｰ 入り端
      LD      Y2E3  ; 締め部　ﾘﾀｰﾝｽﾄｯﾊﾟｰ 抜き SOL
      ANI     X2A5  ; 締め部　ﾘﾀｰﾝｽﾄｯﾊﾟｰ 抜き端
      ORB
      LD      T61  ; 締め部　ﾘﾀｰﾝｽﾄｯﾊﾟｰ 動作異常
      ANI     M20  ; 異常リセット
      ORB
      OUT     T61 K50  ; 締め部　ﾘﾀｰﾝｽﾄｯﾊﾟｰ 動作異常
605   LD      Y2E6  ; 締め部　ﾘﾌﾀｰ 上昇SOL
      ANI     X2AB  ; 締め部　ﾘﾌﾀｰ 　　上昇端
      LD      Y2E7  ; 締め部　ﾘﾌﾀｰ 下降SOL
      ANI     X2AC  ; 締め部　ﾘﾌﾀｰ 　　下降端
      ORB
      LD      T62  ; 締め部 ﾘﾌﾀｰ 動作異常
      ANI     M20  ; 異常リセット
      ORB
      OUT     T62 K100  ; 締め部 ﾘﾌﾀｰ 動作異常
617   LD      Y2E8  ; 締め部　着座確認前進 SOL
      ANI     X2C0  ; 締め部 着座確認 前進端
      LD      Y2E9  ; 締め部　着座確認後退 SOL
      ANI     X2C1  ; 締め部 着座確認 後退端
      ORB
      LD      T63  ; 締め部　着座確認　動作異常
      ANI     M20  ; 異常リセット
      ORB
      OUT     T63 K50  ; 締め部　着座確認　動作異常
629   LD      L156  ; ﾅｯﾄﾗﾝﾅ　締め確認
      AND     M286  ; 締め部　着座確認前進端
      AND     M274  ; 締め部　位置決め 入り端
      AND     Y2EA  ; 締め部　着座確認 SOL
      AND     M13  ; 着座有効
      ANI     L153  ; ﾊﾟﾚｯﾄ着座確認
      AND     T226  ; 締め部　ﾅｯﾄﾗﾝﾅｰ ﾊﾟﾚｯﾄ有り
      OUT     T55 K20  ; ﾊﾟﾚｯﾄ着座異常
640   LD      T55  ; ﾊﾟﾚｯﾄ着座異常
      OUT     C1 K1  ; ﾊﾟﾚｯﾄ着座異常
645   LD      L153  ; ﾊﾟﾚｯﾄ着座確認
      ANI     C1  ; ﾊﾟﾚｯﾄ着座異常
      LD      M20  ; 異常リセット
      AND     C1  ; ﾊﾟﾚｯﾄ着座異常
      ORB
      RST     C1  ; ﾊﾟﾚｯﾄ着座異常
654   LD      L155  ; IAI締め部ﾜｰｸｾｯﾄ　完了
      ANI     L156  ; ﾅｯﾄﾗﾝﾅ　締め確認
      AND     T226  ; 締め部　ﾅｯﾄﾗﾝﾅｰ ﾊﾟﾚｯﾄ有り
      AND     M286  ; 締め部　着座確認前進端
      AND     M274  ; 締め部　位置決め 入り端
      AND     Y2EA  ; 締め部　着座確認 SOL
      AND     M13  ; 着座有効
      ANI     L154  ; 着座つまり検知
      OUT     T57 K50  ; 着座つまり検知
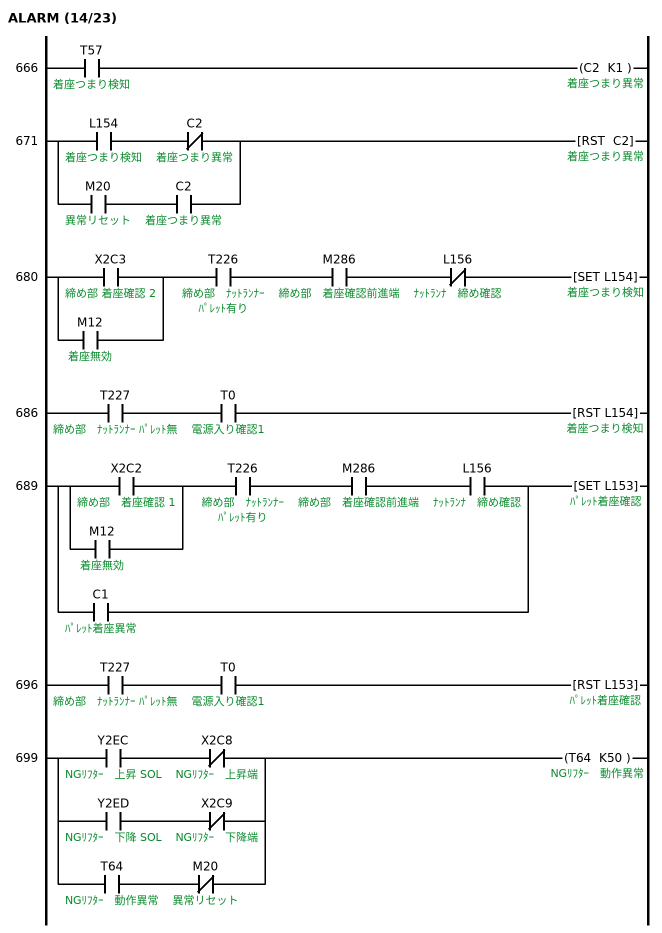
666   LD      T57  ; 着座つまり検知
      OUT     C2 K1  ; 着座つまり異常
671   LD      L154  ; 着座つまり検知
      ANI     C2  ; 着座つまり異常
      LD      M20  ; 異常リセット
      AND     C2  ; 着座つまり異常
      ORB
      RST     C2  ; 着座つまり異常
680   LD      X2C3  ; 締め部 着座確認 2
      OR      M12  ; 着座無効
      AND     T226  ; 締め部　ﾅｯﾄﾗﾝﾅｰ ﾊﾟﾚｯﾄ有り
      AND     M286  ; 締め部　着座確認前進端
      ANI     L156  ; ﾅｯﾄﾗﾝﾅ　締め確認
      SET     L154  ; 着座つまり検知
686   LD      T227  ; 締め部　ﾅｯﾄﾗﾝﾅｰ ﾊﾟﾚｯﾄ無
      AND     T0  ; 電源入り確認1
      RST     L154  ; 着座つまり検知
689   LD      X2C2  ; 締め部　着座確認 1
      OR      M12  ; 着座無効
      AND     T226  ; 締め部　ﾅｯﾄﾗﾝﾅｰ ﾊﾟﾚｯﾄ有り
      AND     M286  ; 締め部　着座確認前進端
      AND     L156  ; ﾅｯﾄﾗﾝﾅ　締め確認
      OR      C1  ; ﾊﾟﾚｯﾄ着座異常
      SET     L153  ; ﾊﾟﾚｯﾄ着座確認
696   LD      T227  ; 締め部　ﾅｯﾄﾗﾝﾅｰ ﾊﾟﾚｯﾄ無
      AND     T0  ; 電源入り確認1
      RST     L153  ; ﾊﾟﾚｯﾄ着座確認
699   LD      Y2EC  ; NGﾘﾌﾀｰ　上昇 SOL
      ANI     X2C8  ; NGﾘﾌﾀｰ　上昇端
      LD      Y2ED  ; NGﾘﾌﾀｰ　下降 SOL
      ANI     X2C9  ; NGﾘﾌﾀｰ　下降端
      ORB
      LD      T64  ; NGﾘﾌﾀｰ　動作異常
      ANI     M20  ; 異常リセット
      ORB
      OUT     T64 K50  ; NGﾘﾌﾀｰ　動作異常
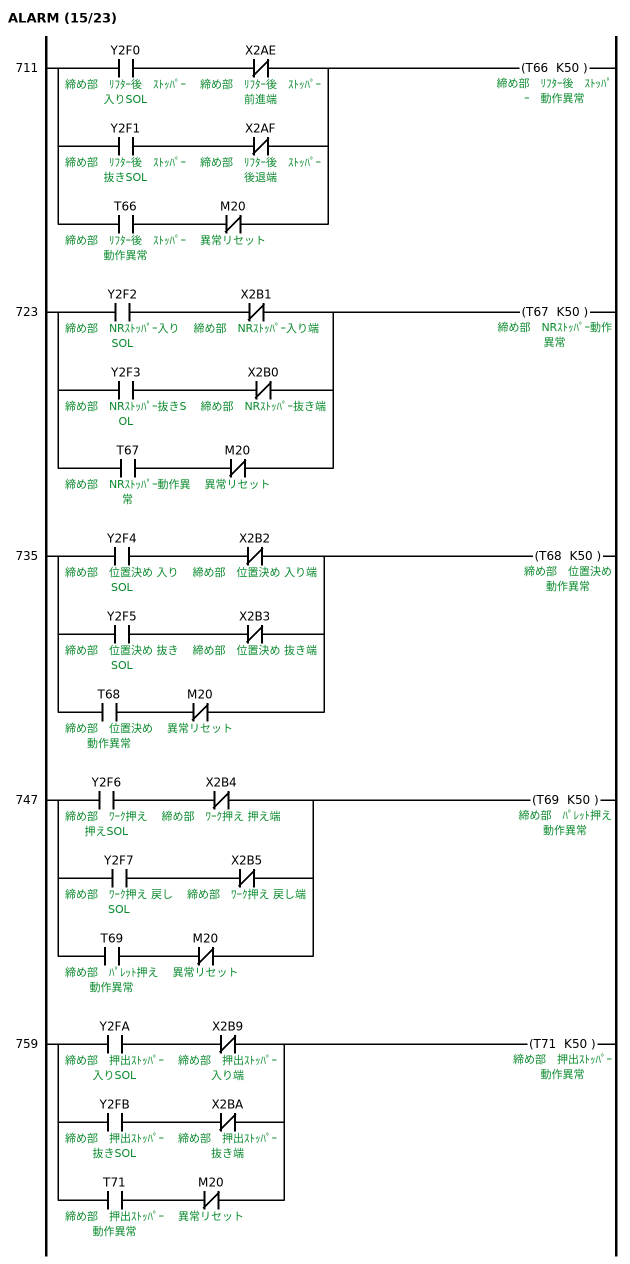
711   LD      Y2F0  ; 締め部　ﾘﾌﾀｰ後　ｽﾄｯﾊﾟｰ　入りSOL
      ANI     X2AE  ; 締め部　ﾘﾌﾀｰ後　ｽﾄｯﾊﾟｰ　前進端
      LD      Y2F1  ; 締め部　ﾘﾌﾀｰ後　ｽﾄｯﾊﾟｰ　抜きSOL
      ANI     X2AF  ; 締め部　ﾘﾌﾀｰ後　ｽﾄｯﾊﾟｰ　後退端
      ORB
      LD      T66  ; 締め部　ﾘﾌﾀｰ後　ｽﾄｯﾊﾟｰ　動作異常
      ANI     M20  ; 異常リセット
      ORB
      OUT     T66 K50  ; 締め部　ﾘﾌﾀｰ後　ｽﾄｯﾊﾟｰ　動作異常
723   LD      Y2F2  ; 締め部　NRｽﾄｯﾊﾟｰ入り SOL
      ANI     X2B1  ; 締め部　NRｽﾄｯﾊﾟｰ入り端
      LD      Y2F3  ; 締め部　NRｽﾄｯﾊﾟｰ抜きSOL
      ANI     X2B0  ; 締め部　NRｽﾄｯﾊﾟｰ抜き端
      ORB
      LD      T67  ; 締め部　NRｽﾄｯﾊﾟｰ動作異常
      ANI     M20  ; 異常リセット
      ORB
      OUT     T67 K50  ; 締め部　NRｽﾄｯﾊﾟｰ動作異常
735   LD      Y2F4  ; 締め部　位置決め 入り SOL
      ANI     X2B2  ; 締め部　位置決め 入り端
      LD      Y2F5  ; 締め部　位置決め 抜き SOL
      ANI     X2B3  ; 締め部　位置決め 抜き端
      ORB
      LD      T68  ; 締め部　位置決め 動作異常
      ANI     M20  ; 異常リセット
      ORB
      OUT     T68 K50  ; 締め部　位置決め 動作異常
747   LD      Y2F6  ; 締め部　ﾜｰｸ押え 押えSOL
      ANI     X2B4  ; 締め部　ﾜｰｸ押え 押え端
      LD      Y2F7  ; 締め部　ﾜｰｸ押え 戻し SOL
      ANI     X2B5  ; 締め部　ﾜｰｸ押え 戻し端
      ORB
      LD      T69  ; 締め部　ﾊﾟﾚｯﾄ押え 動作異常
      ANI     M20  ; 異常リセット
      ORB
      OUT     T69 K50  ; 締め部　ﾊﾟﾚｯﾄ押え 動作異常
759   LD      Y2FA  ; 締め部　押出ｽﾄｯﾊﾟｰ 入りSOL
      ANI     X2B9  ; 締め部　押出ｽﾄｯﾊﾟｰ 入り端
      LD      Y2FB  ; 締め部　押出ｽﾄｯﾊﾟｰ 抜きSOL
      ANI     X2BA  ; 締め部　押出ｽﾄｯﾊﾟｰ 抜き端
      ORB
      LD      T71  ; 締め部　押出ｽﾄｯﾊﾟｰ 動作異常
      ANI     M20  ; 異常リセット
      ORB
      OUT     T71 K50  ; 締め部　押出ｽﾄｯﾊﾟｰ 動作異常
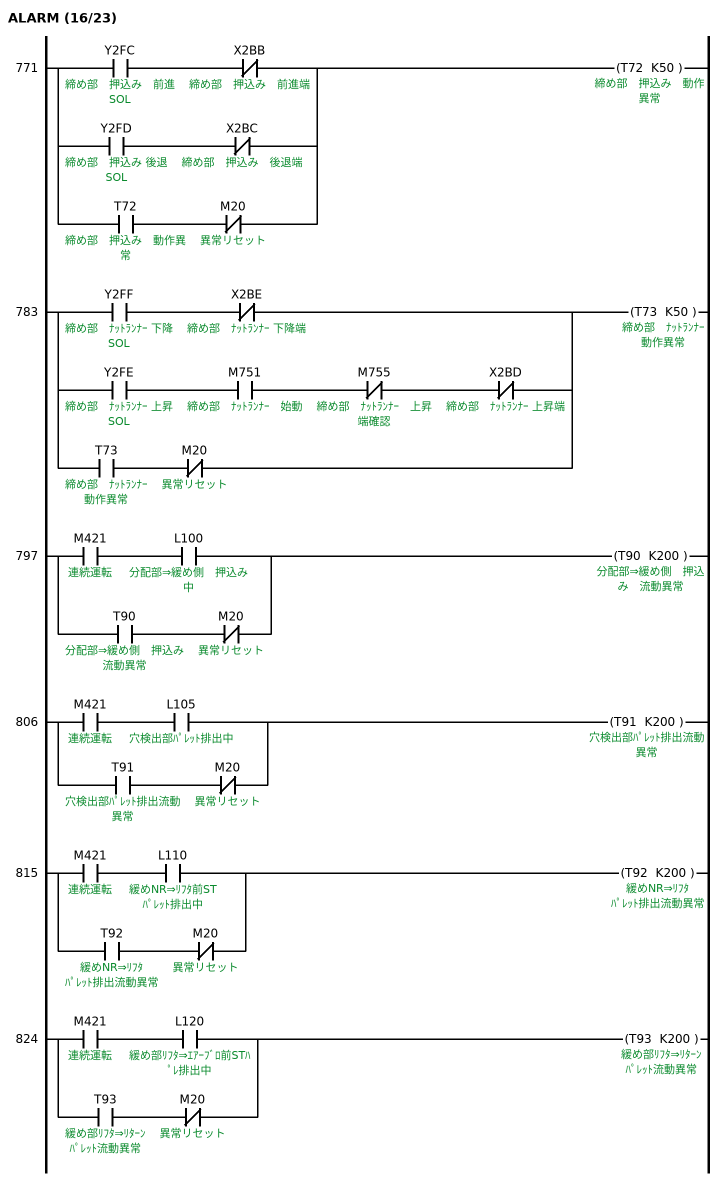
771   LD      Y2FC  ; 締め部　押込み　前進 SOL
      ANI     X2BB  ; 締め部　押込み　前進端
      LD      Y2FD  ; 締め部　押込み 後退 SOL
      ANI     X2BC  ; 締め部　押込み　後退端
      ORB
      LD      T72  ; 締め部　押込み　動作異常
      ANI     M20  ; 異常リセット
      ORB
      OUT     T72 K50  ; 締め部　押込み　動作異常
783   LD      Y2FF  ; 締め部　ﾅｯﾄﾗﾝﾅｰ 下降 SOL
      ANI     X2BE  ; 締め部　ﾅｯﾄﾗﾝﾅｰ 下降端
      LD      Y2FE  ; 締め部　ﾅｯﾄﾗﾝﾅｰ 上昇 SOL
      AND     M751  ; 締め部　ﾅｯﾄﾗﾝﾅｰ　始動
      ANI     M755  ; 締め部　ﾅｯﾄﾗﾝﾅｰ　上昇端確認
      ANI     X2BD  ; 締め部　ﾅｯﾄﾗﾝﾅｰ 上昇端
      ORB
      LD      T73  ; 締め部　ﾅｯﾄﾗﾝﾅｰ 動作異常
      ANI     M20  ; 異常リセット
      ORB
      OUT     T73 K50  ; 締め部　ﾅｯﾄﾗﾝﾅｰ 動作異常
797   LD      M421  ; 連続運転
      AND     L100  ; 分配部⇒緩め側　押込み中
      LD      T90  ; 分配部⇒緩め側　押込み　流動異常
      ANI     M20  ; 異常リセット
      ORB
      OUT     T90 K200  ; 分配部⇒緩め側　押込み　流動異常
806   LD      M421  ; 連続運転
      AND     L105  ; 穴検出部ﾊﾟﾚｯﾄ排出中
      LD      T91  ; 穴検出部ﾊﾟﾚｯﾄ排出流動異常
      ANI     M20  ; 異常リセット
      ORB
      OUT     T91 K200  ; 穴検出部ﾊﾟﾚｯﾄ排出流動異常
815   LD      M421  ; 連続運転
      AND     L110  ; 緩めNR⇒ﾘﾌﾀ前ST ﾊﾟﾚｯﾄ排出中
      LD      T92  ; 緩めNR⇒ﾘﾌﾀ ﾊﾟﾚｯﾄ排出流動異常
      ANI     M20  ; 異常リセット
      ORB
      OUT     T92 K200  ; 緩めNR⇒ﾘﾌﾀ ﾊﾟﾚｯﾄ排出流動異常
824   LD      M421  ; 連続運転
      AND     L120  ; 緩め部ﾘﾌﾀ⇒ｴｱｰﾌﾞﾛ前STﾊﾟﾚ排出中
      LD      T93  ; 緩め部ﾘﾌﾀ⇒ﾘﾀｰﾝ ﾊﾟﾚｯﾄ流動異常
      ANI     M20  ; 異常リセット
      ORB
      OUT     T93 K200  ; 緩め部ﾘﾌﾀ⇒ﾘﾀｰﾝ ﾊﾟﾚｯﾄ流動異常
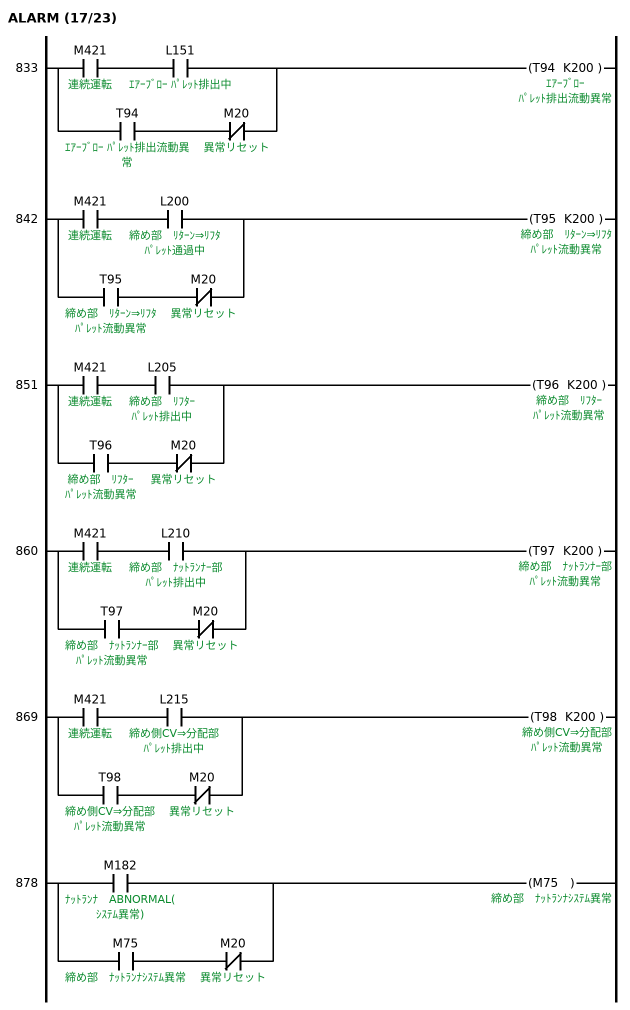
833   LD      M421  ; 連続運転
      AND     L151  ; ｴｱｰﾌﾞﾛｰ ﾊﾟﾚｯﾄ排出中
      LD      T94  ; ｴｱｰﾌﾞﾛｰ ﾊﾟﾚｯﾄ排出流動異常
      ANI     M20  ; 異常リセット
      ORB
      OUT     T94 K200  ; ｴｱｰﾌﾞﾛｰ ﾊﾟﾚｯﾄ排出流動異常
842   LD      M421  ; 連続運転
      AND     L200  ; 締め部　ﾘﾀｰﾝ⇒ﾘﾌﾀ ﾊﾟﾚｯﾄ通過中
      LD      T95  ; 締め部　ﾘﾀｰﾝ⇒ﾘﾌﾀ ﾊﾟﾚｯﾄ流動異常
      ANI     M20  ; 異常リセット
      ORB
      OUT     T95 K200  ; 締め部　ﾘﾀｰﾝ⇒ﾘﾌﾀ ﾊﾟﾚｯﾄ流動異常
851   LD      M421  ; 連続運転
      AND     L205  ; 締め部　ﾘﾌﾀｰ ﾊﾟﾚｯﾄ排出中
      LD      T96  ; 締め部　ﾘﾌﾀｰ ﾊﾟﾚｯﾄ流動異常
      ANI     M20  ; 異常リセット
      ORB
      OUT     T96 K200  ; 締め部　ﾘﾌﾀｰ ﾊﾟﾚｯﾄ流動異常
860   LD      M421  ; 連続運転
      AND     L210  ; 締め部　ﾅｯﾄﾗﾝﾅｰ部 ﾊﾟﾚｯﾄ排出中
      LD      T97  ; 締め部　ﾅｯﾄﾗﾝﾅｰ部 ﾊﾟﾚｯﾄ流動異常
      ANI     M20  ; 異常リセット
      ORB
      OUT     T97 K200  ; 締め部　ﾅｯﾄﾗﾝﾅｰ部 ﾊﾟﾚｯﾄ流動異常
869   LD      M421  ; 連続運転
      AND     L215  ; 締め側CV⇒分配部 ﾊﾟﾚｯﾄ排出中
      LD      T98  ; 締め側CV⇒分配部 ﾊﾟﾚｯﾄ流動異常
      ANI     M20  ; 異常リセット
      ORB
      OUT     T98 K200  ; 締め側CV⇒分配部 ﾊﾟﾚｯﾄ流動異常
878   LD      M182  ; ﾅｯﾄﾗﾝﾅ　ABNORMAL(ｼｽﾃﾑ異常)
      LD      M75  ; 締め部　ﾅｯﾄﾗﾝﾅｼｽﾃﾑ異常
      ANI     M20  ; 異常リセット
      ORB
      OUT     M75  ; 締め部　ﾅｯﾄﾗﾝﾅｼｽﾃﾑ異常
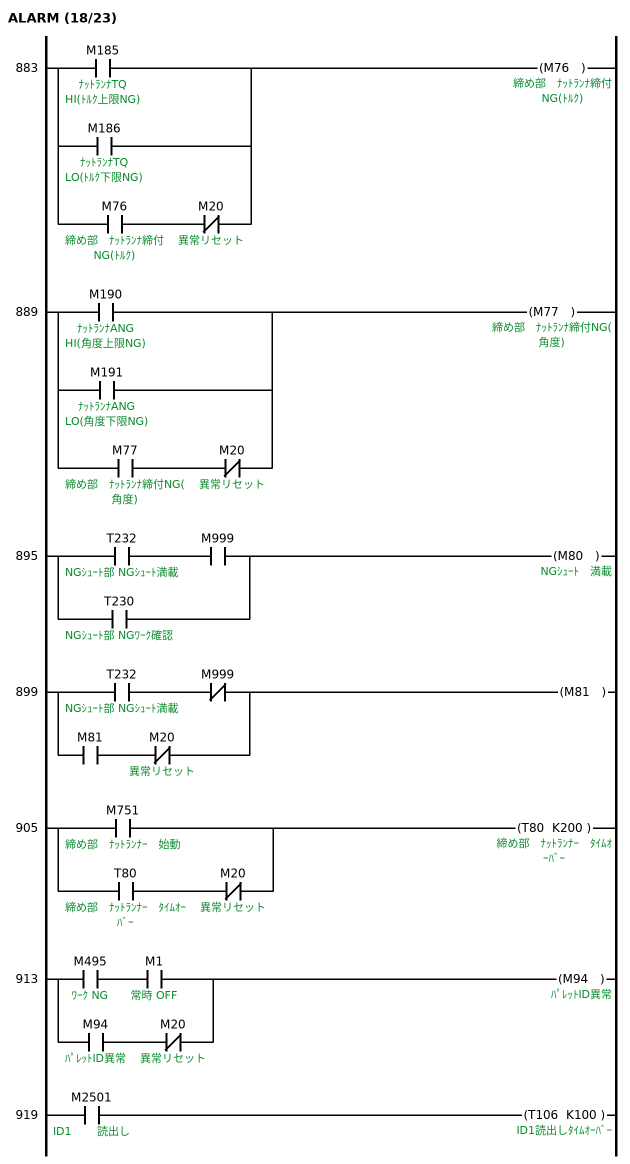
883   LD      M185  ; ﾅｯﾄﾗﾝﾅTQ HI(ﾄﾙｸ上限NG)
      OR      M186  ; ﾅｯﾄﾗﾝﾅTQ LO(ﾄﾙｸ下限NG)
      LD      M76  ; 締め部　ﾅｯﾄﾗﾝﾅ締付 NG(ﾄﾙｸ)
      ANI     M20  ; 異常リセット
      ORB
      OUT     M76  ; 締め部　ﾅｯﾄﾗﾝﾅ締付 NG(ﾄﾙｸ)
889   LD      M190  ; ﾅｯﾄﾗﾝﾅANG HI(角度上限NG)
      OR      M191  ; ﾅｯﾄﾗﾝﾅANG LO(角度下限NG)
      LD      M77  ; 締め部　ﾅｯﾄﾗﾝﾅ締付NG(角度)
      ANI     M20  ; 異常リセット
      ORB
      OUT     M77  ; 締め部　ﾅｯﾄﾗﾝﾅ締付NG(角度)
895   LD      T232  ; NGｼｭｰﾄ部 NGｼｭｰﾄ満載
      AND     M999
      OR      T230  ; NGｼｭｰﾄ部 NGﾜｰｸ確認
      OUT     M80  ; NGｼｭｰﾄ　満載
899   LD      T232  ; NGｼｭｰﾄ部 NGｼｭｰﾄ満載
      ANI     M999
      LD      M81
      ANI     M20  ; 異常リセット
      ORB
      OUT     M81
905   LD      M751  ; 締め部　ﾅｯﾄﾗﾝﾅｰ　始動
      LD      T80  ; 締め部　ﾅｯﾄﾗﾝﾅｰ　ﾀｲﾑｵｰﾊﾞｰ
      ANI     M20  ; 異常リセット
      ORB
      OUT     T80 K200  ; 締め部　ﾅｯﾄﾗﾝﾅｰ　ﾀｲﾑｵｰﾊﾞｰ
913   LD      M495  ; ﾜｰｸ NG
      AND     M1  ; 常時 OFF
      LD      M94  ; ﾊﾟﾚｯﾄID異常
      ANI     M20  ; 異常リセット
      ORB
      OUT     M94  ; ﾊﾟﾚｯﾄID異常
919   LD      M2501  ; ID1　 　読出し
      OUT     T106 K100  ; ID1読出しﾀｲﾑｵｰﾊﾞｰ
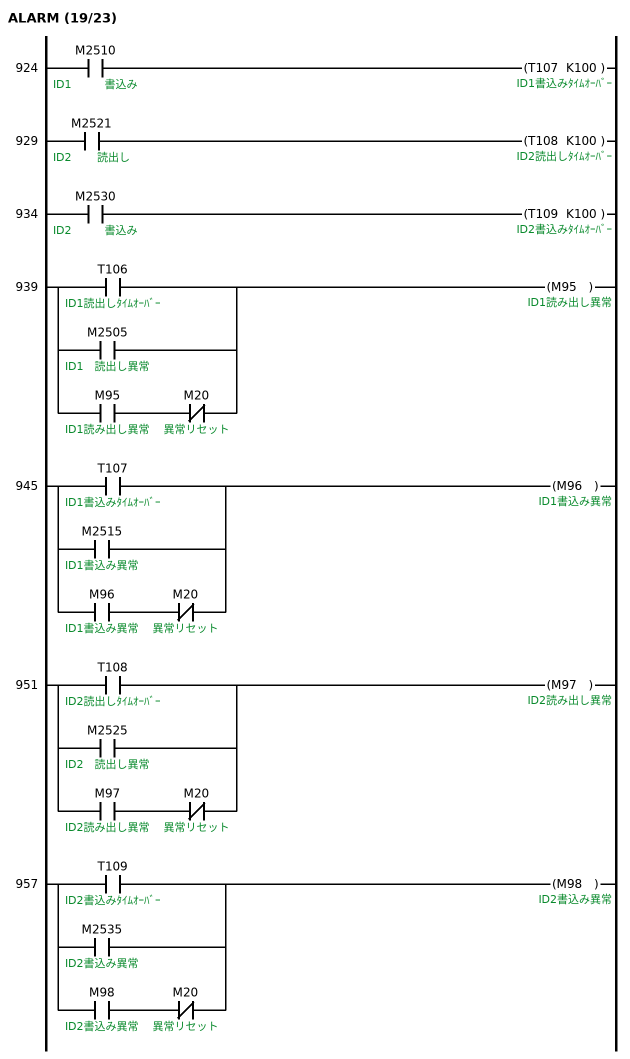
924   LD      M2510  ; ID1　　　書込み
      OUT     T107 K100  ; ID1書込みﾀｲﾑｵｰﾊﾞｰ
929   LD      M2521  ; ID2　 　読出し
      OUT     T108 K100  ; ID2読出しﾀｲﾑｵｰﾊﾞｰ
934   LD      M2530  ; ID2　　　書込み
      OUT     T109 K100  ; ID2書込みﾀｲﾑｵｰﾊﾞｰ
939   LD      T106  ; ID1読出しﾀｲﾑｵｰﾊﾞｰ
      OR      M2505  ; ID1　読出し異常
      LD      M95  ; ID1読み出し異常
      ANI     M20  ; 異常リセット
      ORB
      OUT     M95  ; ID1読み出し異常
945   LD      T107  ; ID1書込みﾀｲﾑｵｰﾊﾞｰ
      OR      M2515  ; ID1書込み異常
      LD      M96  ; ID1書込み異常
      ANI     M20  ; 異常リセット
      ORB
      OUT     M96  ; ID1書込み異常
951   LD      T108  ; ID2読出しﾀｲﾑｵｰﾊﾞｰ
      OR      M2525  ; ID2　読出し異常
      LD      M97  ; ID2読み出し異常
      ANI     M20  ; 異常リセット
      ORB
      OUT     M97  ; ID2読み出し異常
957   LD      T109  ; ID2書込みﾀｲﾑｵｰﾊﾞｰ
      OR      M2535  ; ID2書込み異常
      LD      M98  ; ID2書込み異常
      ANI     M20  ; 異常リセット
      ORB
      OUT     M98  ; ID2書込み異常
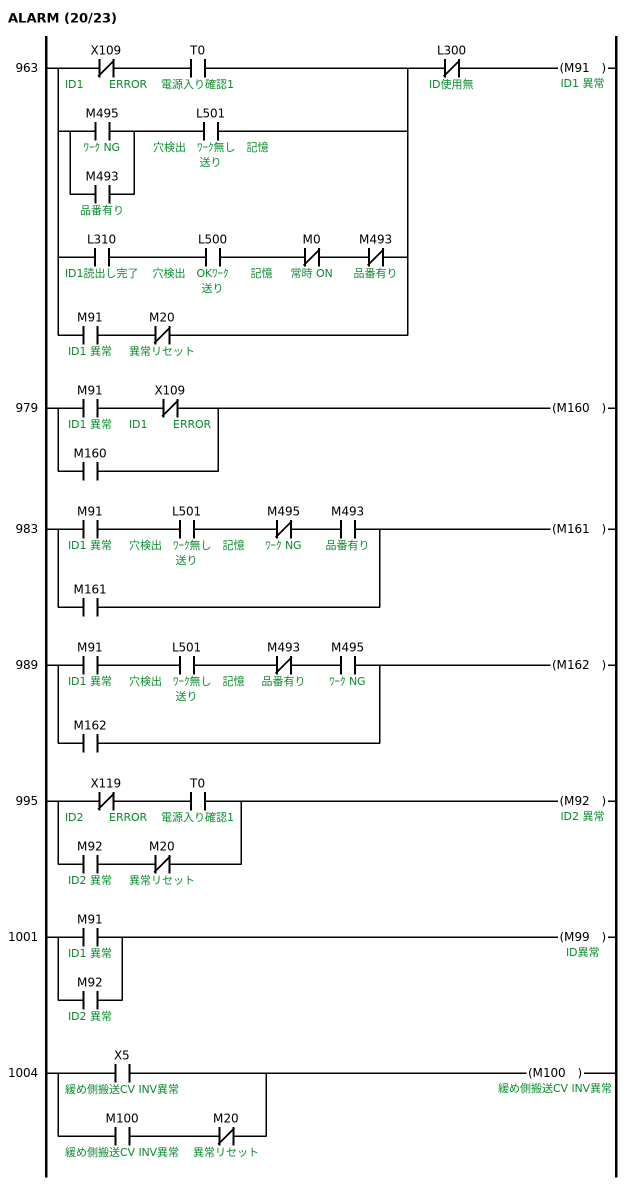
963   LDI     X109  ; ID1　　 ERROR
      AND     T0  ; 電源入り確認1
      LD      M495  ; ﾜｰｸ NG
      OR      M493  ; 品番有り
      AND     L501  ; 穴検出　ﾜｰｸ無し　記憶送り
      ORB
      LD      L310  ; ID1読出し完了
      AND     L500  ; 穴検出　OKﾜｰｸ　　記憶送り
      ANI     M0  ; 常時 ON
      ANI     M493  ; 品番有り
      ORB
      LD      M91  ; ID1 異常
      ANI     M20  ; 異常リセット
      ORB
      ANI     L300  ; ID使用無
      OUT     M91  ; ID1 異常
979   LD      M91  ; ID1 異常
      ANI     X109  ; ID1　　 ERROR
      OR      M160
      OUT     M160
983   LD      M91  ; ID1 異常
      AND     L501  ; 穴検出　ﾜｰｸ無し　記憶送り
      ANI     M495  ; ﾜｰｸ NG
      AND     M493  ; 品番有り
      OR      M161
      OUT     M161
989   LD      M91  ; ID1 異常
      AND     L501  ; 穴検出　ﾜｰｸ無し　記憶送り
      ANI     M493  ; 品番有り
      AND     M495  ; ﾜｰｸ NG
      OR      M162
      OUT     M162
995   LDI     X119  ; ID2　　 ERROR
      AND     T0  ; 電源入り確認1
      LD      M92  ; ID2 異常
      ANI     M20  ; 異常リセット
      ORB
      OUT     M92  ; ID2 異常
1001  LD      M91  ; ID1 異常
      OR      M92  ; ID2 異常
      OUT     M99  ; ID異常
1004  LD      X5  ; 緩め側搬送CV INV異常
      LD      M100  ; 緩め側搬送CV INV異常
      ANI     M20  ; 異常リセット
      ORB
      OUT     M100  ; 緩め側搬送CV INV異常
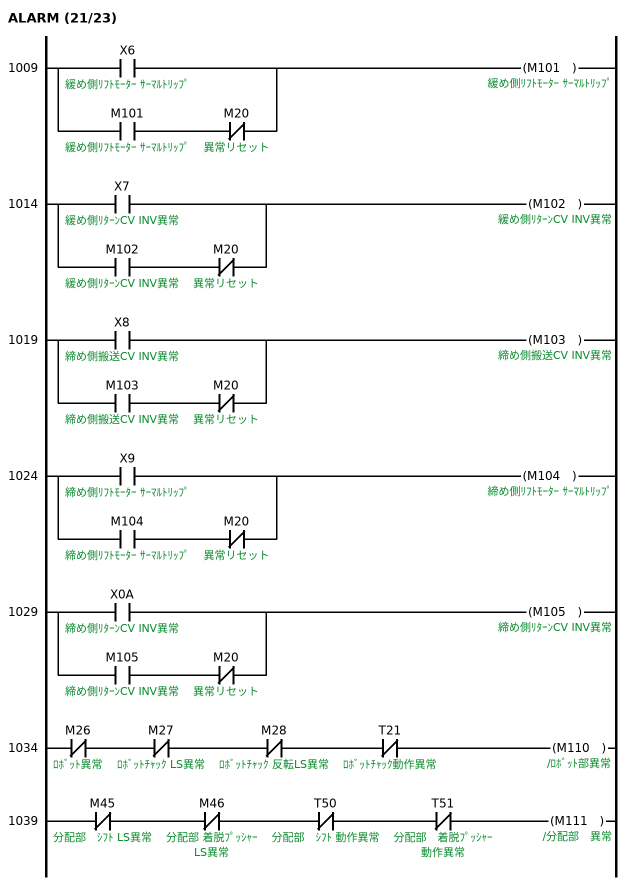
1009  LD      X6  ; 緩め側ﾘﾌﾄﾓｰﾀｰ ｻｰﾏﾙﾄﾘｯﾌﾟ
      LD      M101  ; 緩め側ﾘﾌﾄﾓｰﾀｰ ｻｰﾏﾙﾄﾘｯﾌﾟ
      ANI     M20  ; 異常リセット
      ORB
      OUT     M101  ; 緩め側ﾘﾌﾄﾓｰﾀｰ ｻｰﾏﾙﾄﾘｯﾌﾟ
1014  LD      X7  ; 緩め側ﾘﾀｰﾝCV INV異常
      LD      M102  ; 緩め側ﾘﾀｰﾝCV INV異常
      ANI     M20  ; 異常リセット
      ORB
      OUT     M102  ; 緩め側ﾘﾀｰﾝCV INV異常
1019  LD      X8  ; 締め側搬送CV INV異常
      LD      M103  ; 締め側搬送CV INV異常
      ANI     M20  ; 異常リセット
      ORB
      OUT     M103  ; 締め側搬送CV INV異常
1024  LD      X9  ; 締め側ﾘﾌﾄﾓｰﾀｰ ｻｰﾏﾙﾄﾘｯﾌﾟ
      LD      M104  ; 締め側ﾘﾌﾄﾓｰﾀｰ ｻｰﾏﾙﾄﾘｯﾌﾟ
      ANI     M20  ; 異常リセット
      ORB
      OUT     M104  ; 締め側ﾘﾌﾄﾓｰﾀｰ ｻｰﾏﾙﾄﾘｯﾌﾟ
1029  LD      X0A  ; 締め側ﾘﾀｰﾝCV INV異常
      LD      M105  ; 締め側ﾘﾀｰﾝCV INV異常
      ANI     M20  ; 異常リセット
      ORB
      OUT     M105  ; 締め側ﾘﾀｰﾝCV INV異常
1034  LDI     M26  ; ﾛﾎﾞｯﾄ異常
      ANI     M27  ; ﾛﾎﾞｯﾄﾁｬｯｸ LS異常
      ANI     M28  ; ﾛﾎﾞｯﾄﾁｬｯｸ 反転LS異常
      ANI     T21  ; ﾛﾎﾞｯﾄﾁｬｯｸ動作異常
      OUT     M110  ; /ﾛﾎﾞｯﾄ部異常
1039  LDI     M45  ; 分配部　ｼﾌﾄ LS異常
      ANI     M46  ; 分配部 着脱ﾌﾟｯｼｬｰ LS異常
      ANI     T50  ; 分配部　ｼﾌﾄ 動作異常
      ANI     T51  ; 分配部　着脱ﾌﾟｯｼｬｰ 動作異常
      OUT     M111  ; /分配部　異常
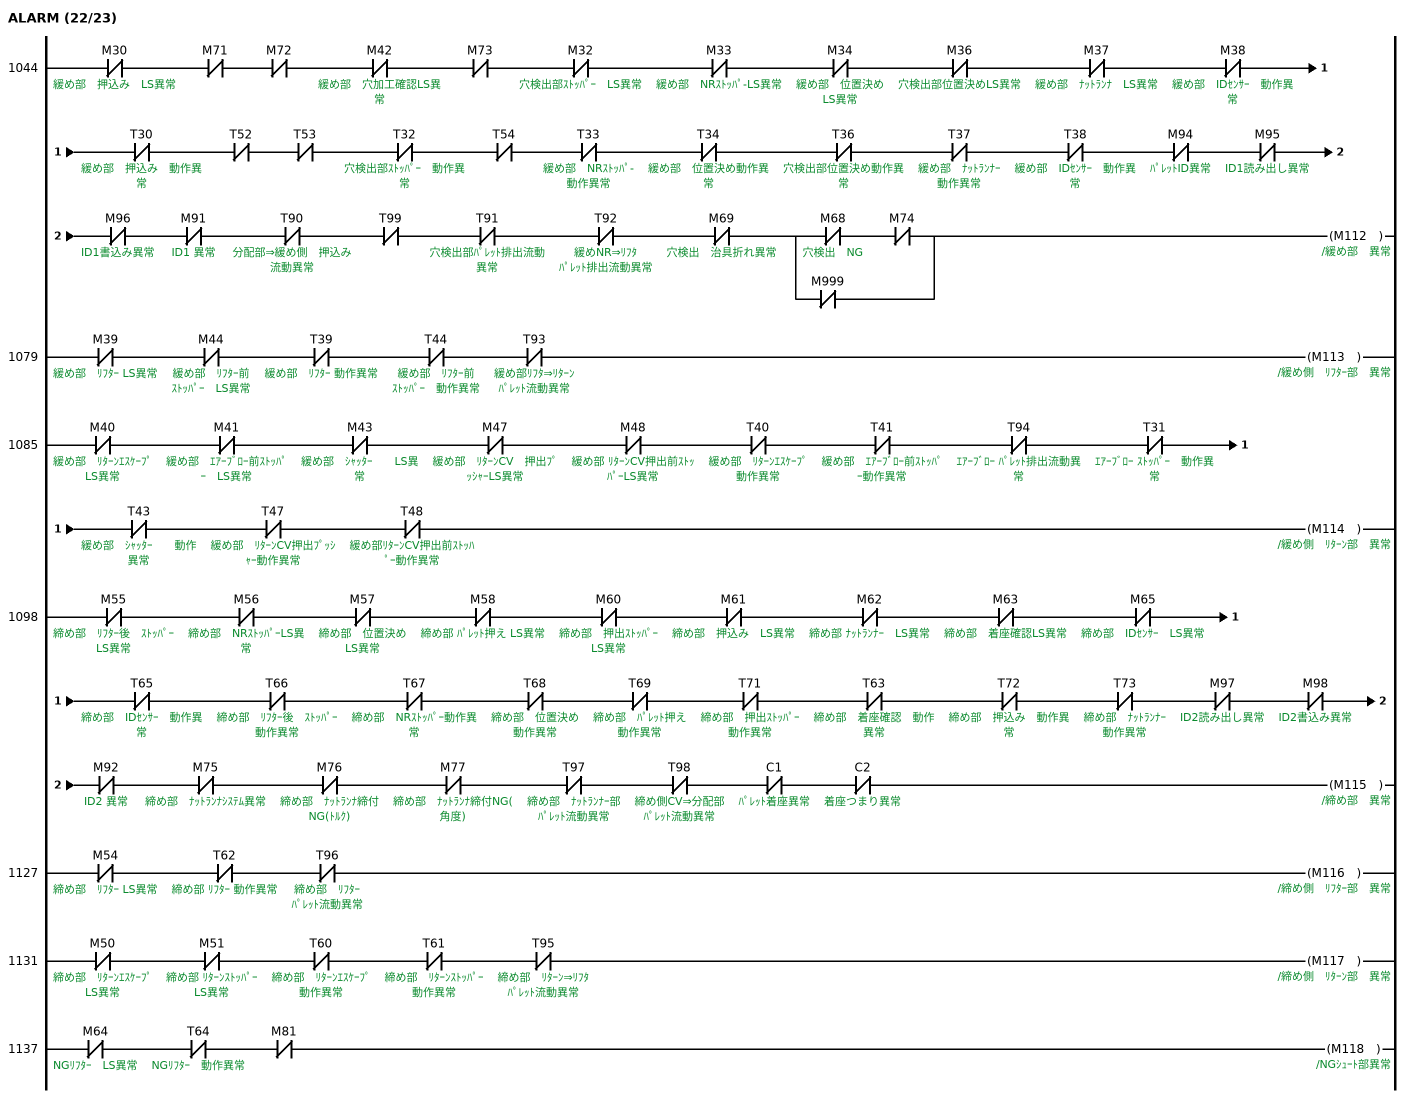
1044  LDI     M30  ; 緩め部　押込み　LS異常
      ANI     M71
      ANI     M72
      ANI     M42  ; 緩め部　穴加工確認LS異常
      ANI     M73
      ANI     M32  ; 穴検出部ｽﾄｯﾊﾟｰ　LS異常
      ANI     M33  ; 緩め部　NRｽﾄｯﾊﾟ-LS異常
      ANI     M34  ; 緩め部　位置決め LS異常
      ANI     M36  ; 穴検出部位置決めLS異常
      ANI     M37  ; 緩め部　ﾅｯﾄﾗﾝﾅ　LS異常
      ANI     M38  ; 緩め部　IDｾﾝｻｰ　動作異常
      ANI     T30  ; 緩め部　押込み　動作異常
      ANI     T52
      ANI     T53
      ANI     T32  ; 穴検出部ｽﾄｯﾊﾟｰ　動作異常
      ANI     T54
      ANI     T33  ; 緩め部　NRｽﾄｯﾊﾟ-動作異常
      ANI     T34  ; 緩め部　位置決め動作異常
      ANI     T36  ; 穴検出部位置決め動作異常
      ANI     T37  ; 緩め部　ﾅｯﾄﾗﾝﾅｰ 動作異常
      ANI     T38  ; 緩め部　IDｾﾝｻｰ　動作異常
      ANI     M94  ; ﾊﾟﾚｯﾄID異常
      ANI     M95  ; ID1読み出し異常
      ANI     M96  ; ID1書込み異常
      ANI     M91  ; ID1 異常
      ANI     T90  ; 分配部⇒緩め側　押込み　流動異常
      ANI     T99
      ANI     T91  ; 穴検出部ﾊﾟﾚｯﾄ排出流動異常
      ANI     T92  ; 緩めNR⇒ﾘﾌﾀ ﾊﾟﾚｯﾄ排出流動異常
      ANI     M69  ; 穴検出　治具折れ異常
      LDI     M68  ; 穴検出　NG
      ANI     M74
      ORI     M999
      ANB
      OUT     M112  ; /緩め部　異常
1079  LDI     M39  ; 緩め部　ﾘﾌﾀｰ LS異常
      ANI     M44  ; 緩め部　ﾘﾌﾀｰ前  ｽﾄｯﾊﾟｰ　LS異常
      ANI     T39  ; 緩め部　ﾘﾌﾀｰ 動作異常
      ANI     T44  ; 緩め部　ﾘﾌﾀｰ前  ｽﾄｯﾊﾟｰ　動作異常
      ANI     T93  ; 緩め部ﾘﾌﾀ⇒ﾘﾀｰﾝ ﾊﾟﾚｯﾄ流動異常
      OUT     M113  ; /緩め側　ﾘﾌﾀｰ部　異常
1085  LDI     M40  ; 緩め部　ﾘﾀｰﾝｴｽｹｰﾌﾟ LS異常
      ANI     M41  ; 緩め部　ｴｱｰﾌﾞﾛｰ前ｽﾄｯﾊﾟｰ　LS異常
      ANI     M43  ; 緩め部　ｼｬｯﾀｰ　　LS異常
      ANI     M47  ; 緩め部　ﾘﾀｰﾝCV　押出ﾌﾟｯｼｬｰLS異常
      ANI     M48  ; 緩め部 ﾘﾀｰﾝCV押出前ｽﾄｯﾊﾟｰLS異常
      ANI     T40  ; 緩め部　ﾘﾀｰﾝｴｽｹｰﾌﾟ 動作異常
      ANI     T41  ; 緩め部　ｴｱｰﾌﾞﾛｰ前ｽﾄｯﾊﾟｰ動作異常
      ANI     T94  ; ｴｱｰﾌﾞﾛｰ ﾊﾟﾚｯﾄ排出流動異常
      ANI     T31  ; ｴｱｰﾌﾞﾛｰ ｽﾄｯﾊﾟｰ　動作異常
      ANI     T43  ; 緩め部　ｼｬｯﾀｰ　　動作異常
      ANI     T47  ; 緩め部　ﾘﾀｰﾝCV押出ﾌﾟｯｼｬｰ動作異常
      ANI     T48  ; 緩め部ﾘﾀｰﾝCV押出前ｽﾄｯﾊﾟｰ動作異常
      OUT     M114  ; /緩め側　ﾘﾀｰﾝ部　異常
1098  LDI     M55  ; 締め部　ﾘﾌﾀｰ後　ｽﾄｯﾊﾟｰ　LS異常
      ANI     M56  ; 締め部　NRｽﾄｯﾊﾟｰLS異常
      ANI     M57  ; 締め部　位置決め LS異常
      ANI     M58  ; 締め部 ﾊﾟﾚｯﾄ押え LS異常
      ANI     M60  ; 締め部　押出ｽﾄｯﾊﾟｰ LS異常
      ANI     M61  ; 締め部　押込み　LS異常
      ANI     M62  ; 締め部 ﾅｯﾄﾗﾝﾅｰ　LS異常
      ANI     M63  ; 締め部　着座確認LS異常
      ANI     M65  ; 締め部　IDｾﾝｻｰ　LS異常
      ANI     T65  ; 締め部　IDｾﾝｻｰ　動作異常
      ANI     T66  ; 締め部　ﾘﾌﾀｰ後　ｽﾄｯﾊﾟｰ　動作異常
      ANI     T67  ; 締め部　NRｽﾄｯﾊﾟｰ動作異常
      ANI     T68  ; 締め部　位置決め 動作異常
      ANI     T69  ; 締め部　ﾊﾟﾚｯﾄ押え 動作異常
      ANI     T71  ; 締め部　押出ｽﾄｯﾊﾟｰ 動作異常
      ANI     T63  ; 締め部　着座確認　動作異常
      ANI     T72  ; 締め部　押込み　動作異常
      ANI     T73  ; 締め部　ﾅｯﾄﾗﾝﾅｰ 動作異常
      ANI     M97  ; ID2読み出し異常
      ANI     M98  ; ID2書込み異常
      ANI     M92  ; ID2 異常
      ANI     M75  ; 締め部　ﾅｯﾄﾗﾝﾅｼｽﾃﾑ異常
      ANI     M76  ; 締め部　ﾅｯﾄﾗﾝﾅ締付 NG(ﾄﾙｸ)
      ANI     M77  ; 締め部　ﾅｯﾄﾗﾝﾅ締付NG(角度)
      ANI     T97  ; 締め部　ﾅｯﾄﾗﾝﾅｰ部 ﾊﾟﾚｯﾄ流動異常
      ANI     T98  ; 締め側CV⇒分配部 ﾊﾟﾚｯﾄ流動異常
      ANI     C1  ; ﾊﾟﾚｯﾄ着座異常
      ANI     C2  ; 着座つまり異常
      OUT     M115  ; /締め部　異常
1127  LDI     M54  ; 締め部　ﾘﾌﾀｰ LS異常
      ANI     T62  ; 締め部 ﾘﾌﾀｰ 動作異常
      ANI     T96  ; 締め部　ﾘﾌﾀｰ ﾊﾟﾚｯﾄ流動異常
      OUT     M116  ; /締め側　ﾘﾌﾀｰ部　異常
1131  LDI     M50  ; 締め部　ﾘﾀｰﾝｴｽｹｰﾌﾟ LS異常
      ANI     M51  ; 締め部 ﾘﾀｰﾝｽﾄｯﾊﾟｰ LS異常
      ANI     T60  ; 締め部　ﾘﾀｰﾝｴｽｹｰﾌﾟ 動作異常
      ANI     T61  ; 締め部　ﾘﾀｰﾝｽﾄｯﾊﾟｰ 動作異常
      ANI     T95  ; 締め部　ﾘﾀｰﾝ⇒ﾘﾌﾀ ﾊﾟﾚｯﾄ流動異常
      OUT     M117  ; /締め側　ﾘﾀｰﾝ部　異常
1137  LDI     M64  ; NGﾘﾌﾀｰ　LS異常
      ANI     T64  ; NGﾘﾌﾀｰ　動作異常
      ANI     M81
      OUT     M118  ; /NGｼｭｰﾄ部異常
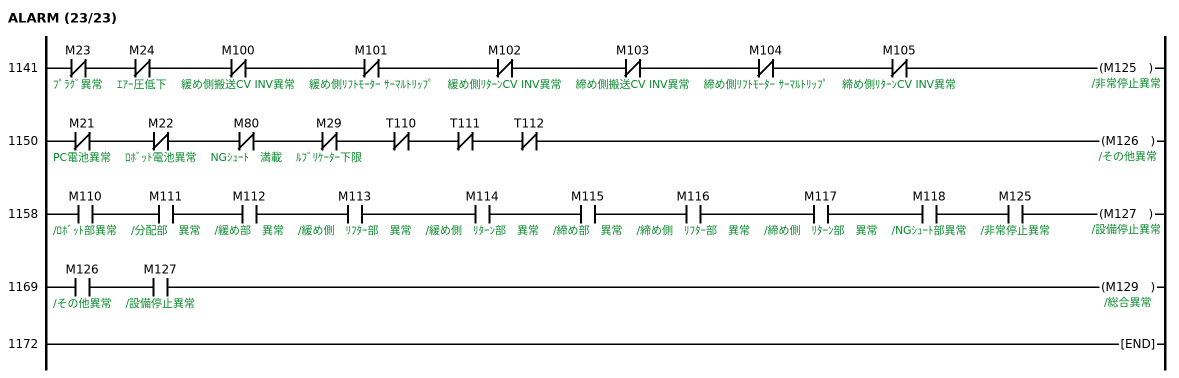
1141  LDI     M23  ; ﾌﾟﾗｸﾞ異常
      ANI     M24  ; ｴｱｰ圧低下
      ANI     M100  ; 緩め側搬送CV INV異常
      ANI     M101  ; 緩め側ﾘﾌﾄﾓｰﾀｰ ｻｰﾏﾙﾄﾘｯﾌﾟ
      ANI     M102  ; 緩め側ﾘﾀｰﾝCV INV異常
      ANI     M103  ; 締め側搬送CV INV異常
      ANI     M104  ; 締め側ﾘﾌﾄﾓｰﾀｰ ｻｰﾏﾙﾄﾘｯﾌﾟ
      ANI     M105  ; 締め側ﾘﾀｰﾝCV INV異常
      OUT     M125  ; /非常停止異常
1150  LDI     M21  ; PC電池異常
      ANI     M22  ; ﾛﾎﾞｯﾄ電池異常
      ANI     M80  ; NGｼｭｰﾄ　満載
      ANI     M29  ; ﾙﾌﾞﾘｹｰﾀｰ下限
      ANI     T110
      ANI     T111
      ANI     T112
      OUT     M126  ; /その他異常
1158  LD      M110  ; /ﾛﾎﾞｯﾄ部異常
      AND     M111  ; /分配部　異常
      AND     M112  ; /緩め部　異常
      AND     M113  ; /緩め側　ﾘﾌﾀｰ部　異常
      AND     M114  ; /緩め側　ﾘﾀｰﾝ部　異常
      AND     M115  ; /締め部　異常
      AND     M116  ; /締め側　ﾘﾌﾀｰ部　異常
      AND     M117  ; /締め側　ﾘﾀｰﾝ部　異常
      AND     M118  ; /NGｼｭｰﾄ部異常
      AND     M125  ; /非常停止異常
      OUT     M127  ; /設備停止異常
1169  LD      M126  ; /その他異常
      AND     M127  ; /設備停止異常
      OUT     M129  ; /総合異常
1172  END
END_PROGRAM
